Yaskawa INFORM job: apremTRJ2.JBI

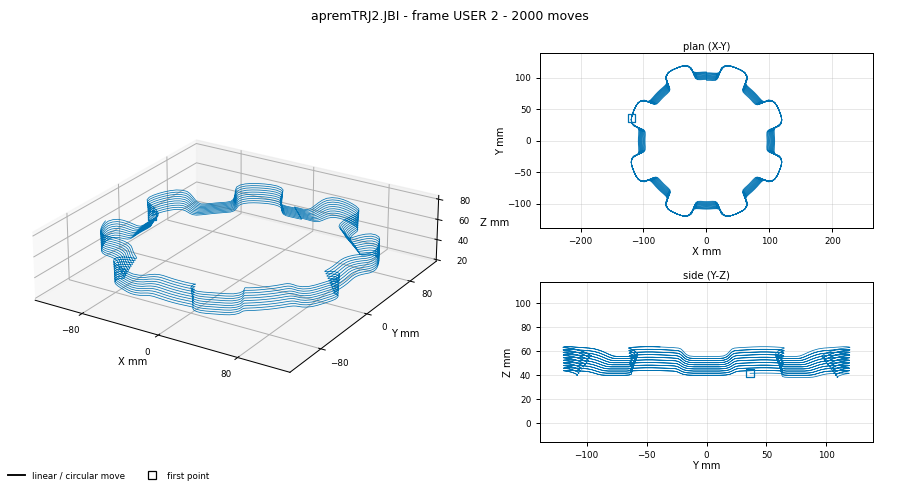
[picture p0: tool path of apremTRJ2.JBI in frame USER 2, 2000 of 2000 moves have a stored position in this frame; points joined in program order, loops and branches not executed]
/JOB
//NAME apremTRJ2
//POS
///NPOS 2000,0,0,0,0,0
///USER 2
///TOOL 1
///POSTYPE USER
///RECTAN
///RCONF 1,0,0,0,0,0,0,0,0,0,0,0,0,0,0,0,0,0,0,0,0,0,0,0
C00000=-119.072,36.353,41.582,179.9283,-0.7231,0.0000
C00001=-118.000,41.045,41.707,179.9989,-0.0034,0.0000
C00002=-116.380,45.594,41.789,179.9994,-0.0015,0.0000
C00003=-114.533,50.053,41.789,179.9993,-0.0015,0.0000
C00004=-112.462,54.416,41.707,179.9984,-0.0032,0.0000
C00005=-109.902,58.491,41.582,179.5393,-0.5620,0.0000
C00006=-106.611,61.626,41.458,179.6621,-0.2455,0.0000
C00007=-103.173,63.375,41.307,179.7307,-0.0735,0.0000
C00008=-100.060,63.578,41.020,-179.7213,-0.0197,0.0000
C00009=-97.017,63.208,40.437,-176.3792,-0.5593,0.0000
C00010=-94.156,62.962,39.673,-168.9691,-0.5777,0.0000
C00011=-91.471,63.401,38.921,-157.5827,5.7610,0.0000
C00012=-88.635,65.218,38.370,-153.3359,22.5360,0.0000
C00013=-85.107,69.037,38.148,-155.1849,27.9206,0.0000
C00014=-81.483,73.239,38.139,-154.7783,27.7766,0.0000
C00015=-77.473,77.473,38.145,-153.4608,26.5387,0.0000
C00016=-73.239,81.483,38.139,-152.2237,25.2220,0.0000
C00017=-69.037,85.107,38.148,-152.0801,24.8157,0.0000
C00018=-65.218,88.635,38.370,-157.4634,26.6637,0.0000
C00019=-63.401,91.471,38.921,-174.2390,22.4173,0.0000
C00020=-62.962,94.156,39.673,179.4223,11.0309,0.0000
C00021=-63.208,97.017,40.437,179.4407,3.6208,0.0000
C00022=-63.578,100.060,41.020,179.9803,0.2787,0.0000
C00023=-63.375,103.173,41.307,179.9265,-0.2693,0.0000
C00024=-61.626,106.611,41.458,179.7545,-0.3379,0.0000
C00025=-58.491,109.902,41.582,179.4380,-0.4607,0.0000
C00026=-54.416,112.462,41.707,179.9968,-0.0016,0.0000
C00027=-50.053,114.533,41.789,179.9985,-0.0007,0.0000
C00028=-45.594,116.380,41.789,179.9985,-0.0006,0.0000
C00029=-41.045,118.000,41.707,179.9966,-0.0011,0.0000
C00030=-36.353,119.072,41.582,179.2769,-0.0717,0.0000
C00031=-31.809,118.962,41.458,179.5875,0.0653,0.0000
C00032=-28.141,117.767,41.307,179.7576,0.1385,0.0000
C00033=-25.796,115.710,41.020,-179.8169,-0.2110,0.0000
C00034=-23.906,113.297,40.437,-177.8329,-2.9566,0.0000
C00035=-22.057,111.099,39.673,-172.5529,-8.2489,0.0000
C00036=-19.849,109.511,38.921,-160.0472,-12.4271,0.0000
C00037=-16.558,108.791,38.370,-147.0366,-3.5281,0.0000
C00038=-11.363,108.997,38.148,-144.9437,2.7334,0.0000
C00039=-5.830,109.405,38.139,-144.7966,2.2545,0.0000
C00040=0.000,109.564,38.145,-144.7664,0.0004,0.0000
C00041=0.000,108.284,39.935,-144.1032,0.0004,0.0000
C00042=5.713,108.130,39.927,-144.1335,-2.3009,0.0000
C00043=11.166,107.733,39.938,-144.2844,-2.6355,0.0000
C00044=16.317,107.567,40.182,-146.6500,4.4566,0.0000
C00045=19.551,108.390,40.791,-161.4224,13.0406,0.0000
C00046=21.713,110.141,41.623,-173.7880,7.6722,0.0000
C00047=23.528,112.556,42.474,-178.5737,2.1635,0.0000
C00048=25.385,115.220,43.124,179.5625,-0.5661,0.0000
C00049=27.691,117.522,43.446,179.0873,-0.5941,0.0000
C00050=31.383,118.911,43.616,179.2076,-0.1524,0.0000
C00051=36.015,119.134,43.755,179.1192,0.0737,0.0000
C00052=40.830,118.071,43.895,179.9841,0.0052,0.0000
C00053=45.521,116.408,43.987,179.9970,0.0012,0.0000
C00054=50.124,114.501,43.987,179.9971,0.0013,0.0000
C00055=54.618,112.360,43.895,179.9851,0.0076,0.0000
C00056=58.774,109.707,43.755,179.3251,0.5708,0.0000
C00057=61.891,106.274,43.616,179.5474,0.6680,0.0000
C00058=63.520,102.681,43.446,179.7747,1.0655,0.0000
C00059=63.523,99.422,43.124,-179.9091,0.7096,0.0000
C00060=62.953,96.226,42.474,179.4782,-2.5377,0.0000
C00061=62.528,93.235,41.623,178.9522,-9.7717,0.0000
C00062=62.818,90.468,40.791,-175.7744,-21.8723,0.0000
C00063=64.524,87.599,40.182,-157.6939,-27.4960,0.0000
C00064=68.283,84.074,39.938,-151.5889,-25.4475,0.0000
C00065=72.420,80.499,39.927,-151.6468,-25.7721,0.0000
C00066=76.568,76.568,39.935,-152.8969,-27.1036,0.0000
C00067=80.499,72.420,39.927,-154.2275,-28.3529,0.0000
C00068=84.074,68.282,39.938,-154.5518,-28.4103,0.0000
C00069=87.599,64.524,40.182,-152.5043,-22.3068,0.0000
C00070=90.468,62.818,40.791,-158.1277,-4.2256,0.0000
C00071=93.235,62.528,41.623,-170.2283,1.0478,0.0000
C00072=96.226,62.953,42.474,-177.4623,0.5218,0.0000
C00073=99.422,63.523,43.124,179.2904,-0.0909,0.0000
C00074=102.681,63.520,43.446,178.9345,0.2253,0.0000
C00075=106.274,61.891,43.616,179.3320,0.4526,0.0000
C00076=109.707,58.774,43.755,179.4292,0.6749,0.0000
C00077=112.360,54.618,43.895,179.9924,0.0149,0.0000
C00078=114.501,50.124,43.987,179.9987,0.0029,0.0000
C00079=116.408,45.521,43.987,179.9988,0.0030,0.0000
C00080=118.071,40.830,43.895,179.9948,0.0159,0.0000
C00081=119.134,36.015,43.755,179.9263,0.8808,0.0000
C00082=118.911,31.383,43.616,-179.8476,0.7924,0.0000
C00083=117.522,27.691,43.446,-179.4059,0.9127,0.0000
C00084=115.220,25.385,43.124,-179.4339,0.4375,0.0000
C00085=112.556,23.528,42.474,177.8365,-1.4263,0.0000
C00086=110.141,21.713,41.623,172.3278,-6.2120,0.0000
C00087=108.390,19.551,40.791,166.9594,-18.5776,0.0000
C00088=107.567,16.317,40.182,175.5434,-33.3500,0.0000
C00089=107.733,11.166,39.938,-177.3645,-35.7156,0.0000
C00090=108.130,5.713,39.927,-177.6991,-35.8665,0.0000
C00091=108.284,0.000,39.935,179.9996,-35.8968,0.0000
C00092=108.130,-5.713,39.927,177.6997,-35.8666,0.0000
C00093=107.733,-11.167,39.938,177.3658,-35.7155,0.0000
C00094=107.567,-16.317,40.182,-175.5442,-33.3502,0.0000
C00095=108.390,-19.551,40.791,-166.9594,-18.5776,0.0000
C00096=110.141,-21.713,41.623,-172.3278,-6.2120,0.0000
C00097=112.556,-23.528,42.474,-177.8365,-1.4263,0.0000
C00098=115.220,-25.385,43.124,179.4339,0.4375,0.0000
C00099=117.522,-27.691,43.446,179.4059,0.9127,0.0000
C00100=118.911,-31.383,43.616,179.8476,0.7924,0.0000
C00101=119.134,-36.015,43.755,-179.9263,0.8808,0.0000
C00102=118.071,-40.830,43.895,-179.9948,0.0159,0.0000
C00103=116.408,-45.521,43.987,-179.9988,0.0030,0.0000
C00104=114.501,-50.124,43.987,-179.9987,0.0029,0.0000
C00105=112.360,-54.618,43.895,-179.9924,0.0149,0.0000
C00106=109.707,-58.774,43.755,-179.4292,0.6749,0.0000
C00107=106.274,-61.891,43.616,-179.3320,0.4526,0.0000
C00108=102.681,-63.520,43.446,-178.9345,0.2253,0.0000
C00109=99.422,-63.523,43.124,-179.2904,-0.0909,0.0000
C00110=96.226,-62.953,42.474,177.4623,0.5218,0.0000
C00111=93.235,-62.528,41.623,170.2283,1.0478,0.0000
C00112=90.468,-62.818,40.791,158.1277,-4.2256,0.0000
C00113=87.599,-64.524,40.182,152.5040,-22.3061,0.0000
C00114=84.074,-68.283,39.938,154.5525,-28.4111,0.0000
C00115=80.499,-72.420,39.927,154.2279,-28.3532,0.0000
C00116=76.568,-76.568,39.935,152.8964,-27.1031,0.0000
C00117=72.420,-80.499,39.927,151.6471,-25.7725,0.0000
C00118=68.282,-84.074,39.938,151.5897,-25.4482,0.0000
C00119=64.524,-87.599,40.182,157.6932,-27.4957,0.0000
C00120=62.818,-90.468,40.791,175.7744,-21.8723,0.0000
C00121=62.528,-93.235,41.623,-178.9522,-9.7717,0.0000
C00122=62.953,-96.226,42.474,-179.4782,-2.5377,0.0000
C00123=63.523,-99.422,43.124,179.9091,0.7096,0.0000
C00124=63.520,-102.681,43.446,-179.7747,1.0655,0.0000
C00125=61.891,-106.274,43.616,-179.5474,0.6680,0.0000
C00126=58.774,-109.707,43.755,-179.3251,0.5708,0.0000
C00127=54.618,-112.360,43.895,-179.9851,0.0076,0.0000
C00128=50.124,-114.501,43.987,-179.9971,0.0013,0.0000
C00129=45.521,-116.408,43.987,-179.9970,0.0012,0.0000
C00130=40.830,-118.071,43.895,-179.9841,0.0052,0.0000
C00131=36.015,-119.134,43.755,-179.1192,0.0737,0.0000
C00132=31.383,-118.911,43.616,-179.2076,-0.1524,0.0000
C00133=27.691,-117.522,43.446,-179.0873,-0.5941,0.0000
C00134=25.385,-115.220,43.124,-179.5625,-0.5661,0.0000
C00135=23.528,-112.556,42.474,178.5737,2.1635,0.0000
C00136=21.713,-110.141,41.623,173.7880,7.6722,0.0000
C00137=19.551,-108.390,40.791,161.4224,13.0406,0.0000
C00138=16.317,-107.567,40.182,146.6500,4.4566,0.0000
C00139=11.166,-107.733,39.938,144.2844,-2.6355,0.0000
C00140=5.713,-108.130,39.927,144.1335,-2.3009,0.0000
C00141=0.000,-108.284,39.935,144.1032,0.0004,0.0000
C00142=0.000,-108.284,39.935,144.1032,0.0004,0.0000
C00143=-5.713,-108.130,39.927,144.1334,2.3003,0.0000
C00144=-11.167,-107.733,39.938,144.2845,2.6342,0.0000
C00145=-16.317,-107.567,40.182,146.6498,-4.4558,0.0000
C00146=-19.551,-108.390,40.791,161.4224,-13.0406,0.0000
C00147=-21.713,-110.141,41.623,173.7880,-7.6722,0.0000
C00148=-23.528,-112.556,42.474,178.5737,-2.1635,0.0000
C00149=-25.385,-115.220,43.124,-179.5625,0.5661,0.0000
C00150=-27.691,-117.522,43.446,-179.0873,0.5941,0.0000
C00151=-31.383,-118.911,43.616,-179.2076,0.1524,0.0000
C00152=-36.015,-119.134,43.755,-179.1192,-0.0737,0.0000
C00153=-40.830,-118.071,43.895,-179.9841,-0.0052,0.0000
C00154=-45.521,-116.408,43.987,-179.9970,-0.0012,0.0000
C00155=-50.124,-114.501,43.987,-179.9971,-0.0013,0.0000
C00156=-54.618,-112.360,43.895,-179.9851,-0.0076,0.0000
C00157=-58.774,-109.707,43.755,-179.3251,-0.5708,0.0000
C00158=-61.891,-106.274,43.616,-179.5474,-0.6680,0.0000
C00159=-63.520,-102.681,43.446,-179.7747,-1.0655,0.0000
C00160=-63.523,-99.422,43.124,179.9091,-0.7096,0.0000
C00161=-62.953,-96.226,42.474,-179.4782,2.5377,0.0000
C00162=-62.528,-93.235,41.623,-178.9522,9.7717,0.0000
C00163=-62.818,-90.468,40.791,175.7744,21.8723,0.0000
C00164=-64.524,-87.599,40.182,157.6939,27.4960,0.0000
C00165=-68.283,-84.074,39.938,151.5889,25.4475,0.0000
C00166=-72.420,-80.499,39.927,151.6468,25.7721,0.0000
C00167=-76.568,-76.568,39.935,152.8969,27.1036,0.0000
C00168=-80.499,-72.420,39.927,154.2275,28.3529,0.0000
C00169=-84.074,-68.282,39.938,154.5518,28.4103,0.0000
C00170=-87.599,-64.524,40.182,152.5043,22.3068,0.0000
C00171=-90.468,-62.818,40.791,158.1277,4.2256,0.0000
C00172=-93.235,-62.528,41.623,170.2283,-1.0478,0.0000
C00173=-96.226,-62.953,42.474,177.4623,-0.5218,0.0000
C00174=-99.422,-63.523,43.124,-179.2904,0.0909,0.0000
C00175=-102.681,-63.520,43.446,-178.9345,-0.2253,0.0000
C00176=-106.274,-61.891,43.616,-179.3320,-0.4526,0.0000
C00177=-109.707,-58.774,43.755,-179.4292,-0.6749,0.0000
C00178=-112.360,-54.618,43.895,-179.9924,-0.0149,0.0000
C00179=-114.501,-50.124,43.987,-179.9987,-0.0029,0.0000
C00180=-116.408,-45.521,43.987,-179.9988,-0.0030,0.0000
C00181=-118.071,-40.830,43.895,-179.9948,-0.0159,0.0000
C00182=-119.134,-36.015,43.755,-179.9263,-0.8808,0.0000
C00183=-118.911,-31.383,43.616,179.8476,-0.7924,0.0000
C00184=-117.522,-27.691,43.446,179.4059,-0.9127,0.0000
C00185=-115.220,-25.385,43.124,179.4339,-0.4375,0.0000
C00186=-112.556,-23.528,42.474,-177.8365,1.4263,0.0000
C00187=-110.141,-21.713,41.623,-172.3278,6.2120,0.0000
C00188=-108.390,-19.551,40.791,-166.9594,18.5776,0.0000
C00189=-107.567,-16.317,40.182,-175.5434,33.3500,0.0000
C00190=-107.733,-11.166,39.938,177.3645,35.7156,0.0000
C00191=-108.130,-5.713,39.927,177.6991,35.8665,0.0000
C00192=-108.284,0.000,39.935,-179.9996,35.8968,0.0000
C00193=-108.130,5.713,39.927,-177.6997,35.8666,0.0000
C00194=-107.733,11.167,39.938,-177.3658,35.7155,0.0000
C00195=-107.567,16.317,40.182,175.5442,33.3502,0.0000
C00196=-108.390,19.551,40.791,166.9594,18.5776,0.0000
C00197=-110.141,21.713,41.623,172.3278,6.2120,0.0000
C00198=-112.556,23.528,42.474,177.8365,1.4263,0.0000
C00199=-115.220,25.385,43.124,-179.4339,-0.4375,0.0000
C00200=-117.522,27.691,43.446,-179.4059,-0.9127,0.0000
C00201=-118.911,31.383,43.616,-179.8476,-0.7924,0.0000
C00202=-119.134,36.015,43.755,179.9263,-0.8808,0.0000
C00203=-118.071,40.830,43.895,179.9948,-0.0159,0.0000
C00204=-116.408,45.521,43.987,179.9988,-0.0030,0.0000
C00205=-114.501,50.124,43.987,179.9987,-0.0029,0.0000
C00206=-112.360,54.618,43.895,179.9924,-0.0149,0.0000
C00207=-109.707,58.774,43.755,179.4292,-0.6749,0.0000
C00208=-106.274,61.891,43.616,179.3320,-0.4526,0.0000
C00209=-102.681,63.520,43.446,178.9345,-0.2253,0.0000
C00210=-99.422,63.523,43.124,179.2904,0.0909,0.0000
C00211=-96.226,62.953,42.474,-177.4623,-0.5218,0.0000
C00212=-93.235,62.528,41.623,-170.2283,-1.0478,0.0000
C00213=-90.468,62.818,40.791,-158.1277,4.2256,0.0000
C00214=-87.599,64.524,40.182,-152.5040,22.3061,0.0000
C00215=-84.074,68.283,39.938,-154.5525,28.4111,0.0000
C00216=-80.499,72.420,39.927,-154.2279,28.3532,0.0000
C00217=-76.568,76.568,39.935,-152.8964,27.1031,0.0000
C00218=-72.420,80.499,39.927,-151.6471,25.7725,0.0000
C00219=-68.282,84.074,39.938,-151.5897,25.4482,0.0000
C00220=-64.524,87.599,40.182,-157.6932,27.4957,0.0000
C00221=-62.818,90.468,40.791,-175.7744,21.8723,0.0000
C00222=-62.528,93.235,41.623,178.9522,9.7717,0.0000
C00223=-62.953,96.226,42.474,179.4782,2.5377,0.0000
C00224=-63.523,99.422,43.124,-179.9091,-0.7096,0.0000
C00225=-63.520,102.681,43.446,179.7747,-1.0655,0.0000
C00226=-61.891,106.274,43.616,179.5474,-0.6680,0.0000
C00227=-58.774,109.707,43.755,179.3251,-0.5708,0.0000
C00228=-54.618,112.360,43.895,179.9851,-0.0076,0.0000
C00229=-50.124,114.501,43.987,179.9971,-0.0013,0.0000
C00230=-45.521,116.408,43.987,179.9970,-0.0012,0.0000
C00231=-40.830,118.071,43.895,179.9841,-0.0052,0.0000
C00232=-36.015,119.134,43.755,179.1192,-0.0737,0.0000
C00233=-31.383,118.911,43.616,179.2076,0.1524,0.0000
C00234=-27.691,117.522,43.446,179.0873,0.5941,0.0000
C00235=-25.385,115.220,43.124,179.5625,0.5661,0.0000
C00236=-23.528,112.556,42.474,-178.5737,-2.1635,0.0000
C00237=-21.713,110.141,41.623,-173.7880,-7.6722,0.0000
C00238=-19.551,108.390,40.791,-161.4224,-13.0406,0.0000
C00239=-16.317,107.567,40.182,-146.6498,-4.4558,0.0000
C00240=-11.167,107.733,39.938,-144.2845,2.6342,0.0000
C00241=-5.713,108.130,39.927,-144.1334,2.3003,0.0000
C00242=0.000,108.284,39.935,-144.1032,0.0004,0.0000
C00243=0.000,106.985,41.710,-143.5099,0.0004,0.0000
C00244=5.594,106.835,41.702,-143.5401,-2.3406,0.0000
C00245=10.967,106.449,41.714,-143.6958,-2.5164,0.0000
C00246=16.072,106.324,41.981,-146.3715,5.4141,0.0000
C00247=19.249,107.251,42.649,-162.9140,13.4061,0.0000
C00248=21.363,109.167,43.565,-174.8995,6.9770,0.0000
C00249=23.141,111.802,44.504,-179.1921,1.3529,0.0000
C00250=24.965,114.720,45.225,179.0571,-1.3592,0.0000
C00251=27.231,117.271,45.583,178.4751,-1.1175,0.0000
C00252=30.949,118.858,45.772,178.8291,-0.2647,0.0000
C00253=35.669,119.197,45.927,178.9615,0.0712,0.0000
C00254=40.611,118.143,46.083,179.9716,0.0092,0.0000
C00255=45.447,116.436,46.186,179.9955,0.0017,0.0000
C00256=50.197,114.469,46.186,179.9956,0.0019,0.0000
C00257=54.824,112.256,46.083,179.9734,0.0136,0.0000
C00258=59.063,109.507,45.927,179.2153,0.6841,0.0000
C00259=62.161,105.930,45.772,179.3591,1.0151,0.0000
C00260=63.668,102.179,45.583,179.7118,1.8682,0.0000
C00261=63.466,98.772,45.225,-179.7055,1.6276,0.0000
C00262=62.692,95.419,44.504,179.6145,-1.5278,0.0000
C00263=62.087,92.299,43.565,178.6584,-8.5110,0.0000
C00264=62.227,89.449,42.649,-177.2056,-21.1007,0.0000
C00265=63.818,86.547,41.981,-158.0362,-28.2502,0.0000
C00266=67.516,83.026,41.714,-151.1639,-26.0321,0.0000
C00267=71.588,79.499,41.702,-151.1291,-26.2693,0.0000
C00268=75.650,75.650,41.710,-152.3887,-27.6118,0.0000
C00269=79.499,71.588,41.702,-153.7304,-28.8707,0.0000
C00270=83.026,67.516,41.714,-153.9672,-28.8353,0.0000
C00271=86.547,63.818,41.981,-151.7501,-21.9645,0.0000
C00272=89.449,62.227,42.649,-158.8993,-2.7944,0.0000
C00273=92.299,62.087,43.565,-171.4890,1.3416,0.0000
C00274=95.419,62.692,44.504,-178.4722,0.3855,0.0000
C00275=98.772,63.466,45.225,178.3724,-0.2945,0.0000
C00276=102.179,63.668,45.583,178.1318,0.2882,0.0000
C00277=105.930,62.161,45.772,178.9849,0.6409,0.0000
C00278=109.507,59.063,45.927,179.3159,0.7847,0.0000
C00279=112.256,54.824,46.083,179.9864,0.0266,0.0000
C00280=114.469,50.197,46.186,179.9981,0.0044,0.0000
C00281=116.436,45.447,46.186,179.9983,0.0045,0.0000
C00282=118.143,40.611,46.083,179.9908,0.0284,0.0000
C00283=119.197,35.669,45.927,179.9288,1.0385,0.0000
C00284=118.858,30.949,45.772,-179.7353,1.1709,0.0000
C00285=117.271,27.231,45.583,-178.8825,1.5249,0.0000
C00286=114.720,24.965,45.225,-178.6408,0.9429,0.0000
C00287=111.802,23.141,44.504,178.6471,-0.8079,0.0000
C00288=109.167,21.363,43.565,173.0230,-5.1005,0.0000
C00289=107.251,19.249,42.649,166.5939,-17.0860,0.0000
C00290=106.324,16.072,41.981,174.5859,-33.6285,0.0000
C00291=106.449,10.967,41.714,-177.4836,-36.3042,0.0000
C00292=106.835,5.594,41.702,-177.6594,-36.4599,0.0000
C00293=106.985,0.000,41.710,179.9996,-36.4901,0.0000
C00294=106.835,-5.594,41.702,177.6600,-36.4599,0.0000
C00295=106.449,-10.967,41.714,177.4851,-36.3040,0.0000
C00296=106.324,-16.072,41.981,-174.5868,-33.6287,0.0000
C00297=107.251,-19.249,42.649,-166.5939,-17.0860,0.0000
C00298=109.167,-21.363,43.565,-173.0230,-5.1005,0.0000
C00299=111.802,-23.141,44.504,-178.6471,-0.8079,0.0000
C00300=114.720,-24.965,45.225,178.6408,0.9429,0.0000
C00301=117.271,-27.231,45.583,178.8825,1.5249,0.0000
C00302=118.858,-30.949,45.772,179.7353,1.1709,0.0000
C00303=119.197,-35.669,45.927,-179.9288,1.0385,0.0000
C00304=118.143,-40.611,46.083,-179.9908,0.0284,0.0000
C00305=116.436,-45.447,46.186,-179.9983,0.0045,0.0000
C00306=114.469,-50.197,46.186,-179.9981,0.0044,0.0000
C00307=112.256,-54.824,46.083,-179.9864,0.0266,0.0000
C00308=109.507,-59.063,45.927,-179.3159,0.7847,0.0000
C00309=105.930,-62.161,45.772,-178.9849,0.6409,0.0000
C00310=102.179,-63.668,45.583,-178.1318,0.2882,0.0000
C00311=98.772,-63.466,45.225,-178.3724,-0.2945,0.0000
C00312=95.419,-62.692,44.504,178.4722,0.3855,0.0000
C00313=92.299,-62.087,43.565,171.4890,1.3416,0.0000
C00314=89.449,-62.227,42.649,158.8993,-2.7944,0.0000
C00315=86.547,-63.818,41.981,151.7498,-21.9638,0.0000
C00316=83.026,-67.516,41.714,153.9679,-28.8361,0.0000
C00317=79.499,-71.588,41.702,153.7307,-28.8709,0.0000
C00318=75.650,-75.650,41.710,152.3882,-27.6113,0.0000
C00319=71.588,-79.499,41.702,151.1293,-26.2696,0.0000
C00320=67.516,-83.026,41.714,151.1647,-26.0328,0.0000
C00321=63.818,-86.547,41.981,158.0355,-28.2499,0.0000
C00322=62.227,-89.449,42.649,177.2056,-21.1007,0.0000
C00323=62.087,-92.299,43.565,-178.6584,-8.5110,0.0000
C00324=62.692,-95.419,44.504,-179.6145,-1.5278,0.0000
C00325=63.466,-98.772,45.225,179.7055,1.6276,0.0000
C00326=63.668,-102.179,45.583,-179.7118,1.8682,0.0000
C00327=62.161,-105.930,45.772,-179.3591,1.0151,0.0000
C00328=59.063,-109.507,45.927,-179.2153,0.6841,0.0000
C00329=54.824,-112.256,46.083,-179.9734,0.0136,0.0000
C00330=50.197,-114.469,46.186,-179.9956,0.0019,0.0000
C00331=45.447,-116.436,46.186,-179.9955,0.0017,0.0000
C00332=40.611,-118.143,46.083,-179.9716,0.0092,0.0000
C00333=35.669,-119.197,45.927,-178.9615,0.0712,0.0000
C00334=30.949,-118.858,45.772,-178.8291,-0.2647,0.0000
C00335=27.231,-117.271,45.583,-178.4751,-1.1175,0.0000
C00336=24.965,-114.720,45.225,-179.0571,-1.3592,0.0000
C00337=23.141,-111.802,44.504,179.1921,1.3529,0.0000
C00338=21.363,-109.167,43.565,174.8995,6.9770,0.0000
C00339=19.249,-107.251,42.649,162.9140,13.4061,0.0000
C00340=16.072,-106.324,41.981,146.3715,5.4141,0.0000
C00341=10.967,-106.449,41.714,143.6958,-2.5164,0.0000
C00342=5.594,-106.835,41.702,143.5401,-2.3406,0.0000
C00343=0.000,-106.985,41.710,143.5099,0.0004,0.0000
C00344=0.000,-106.985,41.710,143.5099,0.0004,0.0000
C00345=-5.594,-106.835,41.702,143.5401,2.3400,0.0000
C00346=-10.967,-106.449,41.714,143.6960,2.5149,0.0000
C00347=-16.072,-106.324,41.981,146.3713,-5.4132,0.0000
C00348=-19.249,-107.251,42.649,162.9140,-13.4061,0.0000
C00349=-21.363,-109.167,43.565,174.8995,-6.9770,0.0000
C00350=-23.141,-111.802,44.504,179.1921,-1.3529,0.0000
C00351=-24.965,-114.720,45.225,-179.0571,1.3592,0.0000
C00352=-27.231,-117.271,45.583,-178.4751,1.1175,0.0000
C00353=-30.949,-118.858,45.772,-178.8291,0.2647,0.0000
C00354=-35.669,-119.197,45.927,-178.9615,-0.0712,0.0000
C00355=-40.611,-118.143,46.083,-179.9716,-0.0092,0.0000
C00356=-45.447,-116.436,46.186,-179.9955,-0.0017,0.0000
C00357=-50.197,-114.469,46.186,-179.9956,-0.0019,0.0000
C00358=-54.824,-112.256,46.083,-179.9734,-0.0136,0.0000
C00359=-59.063,-109.507,45.927,-179.2153,-0.6841,0.0000
C00360=-62.161,-105.930,45.772,-179.3591,-1.0151,0.0000
C00361=-63.668,-102.179,45.583,-179.7118,-1.8682,0.0000
C00362=-63.466,-98.772,45.225,179.7055,-1.6276,0.0000
C00363=-62.692,-95.419,44.504,-179.6145,1.5278,0.0000
C00364=-62.087,-92.299,43.565,-178.6584,8.5110,0.0000
C00365=-62.227,-89.449,42.649,177.2056,21.1007,0.0000
C00366=-63.818,-86.547,41.981,158.0362,28.2502,0.0000
C00367=-67.516,-83.026,41.714,151.1639,26.0321,0.0000
C00368=-71.588,-79.499,41.702,151.1291,26.2693,0.0000
C00369=-75.650,-75.650,41.710,152.3887,27.6118,0.0000
C00370=-79.499,-71.588,41.702,153.7304,28.8707,0.0000
C00371=-83.026,-67.516,41.714,153.9672,28.8353,0.0000
C00372=-86.547,-63.818,41.981,151.7501,21.9645,0.0000
C00373=-89.449,-62.227,42.649,158.8993,2.7944,0.0000
C00374=-92.299,-62.087,43.565,171.4890,-1.3416,0.0000
C00375=-95.419,-62.692,44.504,178.4722,-0.3855,0.0000
C00376=-98.772,-63.466,45.225,-178.3724,0.2945,0.0000
C00377=-102.179,-63.668,45.583,-178.1318,-0.2882,0.0000
C00378=-105.930,-62.161,45.772,-178.9849,-0.6409,0.0000
C00379=-109.507,-59.063,45.927,-179.3159,-0.7847,0.0000
C00380=-112.256,-54.824,46.083,-179.9864,-0.0266,0.0000
C00381=-114.469,-50.197,46.186,-179.9981,-0.0044,0.0000
C00382=-116.436,-45.447,46.186,-179.9983,-0.0045,0.0000
C00383=-118.143,-40.611,46.083,-179.9908,-0.0284,0.0000
C00384=-119.197,-35.669,45.927,-179.9288,-1.0385,0.0000
C00385=-118.858,-30.949,45.772,179.7353,-1.1709,0.0000
C00386=-117.271,-27.231,45.583,178.8825,-1.5249,0.0000
C00387=-114.720,-24.965,45.225,178.6408,-0.9429,0.0000
C00388=-111.802,-23.141,44.504,-178.6471,0.8079,0.0000
C00389=-109.167,-21.363,43.565,-173.0230,5.1005,0.0000
C00390=-107.251,-19.249,42.649,-166.5939,17.0860,0.0000
C00391=-106.324,-16.072,41.981,-174.5859,33.6285,0.0000
C00392=-106.449,-10.967,41.714,177.4836,36.3042,0.0000
C00393=-106.835,-5.594,41.702,177.6594,36.4599,0.0000
C00394=-106.985,0.000,41.710,-179.9996,36.4901,0.0000
C00395=-106.835,5.594,41.702,-177.6600,36.4599,0.0000
C00396=-106.449,10.967,41.714,-177.4851,36.3040,0.0000
C00397=-106.324,16.072,41.981,174.5868,33.6287,0.0000
C00398=-107.251,19.249,42.649,166.5939,17.0860,0.0000
C00399=-109.167,21.363,43.565,173.0230,5.1005,0.0000
C00400=-111.802,23.141,44.504,178.6471,0.8079,0.0000
C00401=-114.720,24.965,45.225,-178.6408,-0.9429,0.0000
C00402=-117.271,27.231,45.583,-178.8825,-1.5249,0.0000
C00403=-118.858,30.949,45.772,-179.7353,-1.1709,0.0000
C00404=-119.197,35.669,45.927,179.9288,-1.0385,0.0000
C00405=-118.143,40.611,46.083,179.9908,-0.0284,0.0000
C00406=-116.436,45.447,46.186,179.9983,-0.0045,0.0000
C00407=-114.469,50.197,46.186,179.9981,-0.0044,0.0000
C00408=-112.256,54.824,46.083,179.9864,-0.0266,0.0000
C00409=-109.507,59.063,45.927,179.3159,-0.7847,0.0000
C00410=-105.930,62.161,45.772,178.9849,-0.6409,0.0000
C00411=-102.179,63.668,45.583,178.1318,-0.2882,0.0000
C00412=-98.772,63.466,45.225,178.3724,0.2945,0.0000
C00413=-95.419,62.692,44.504,-178.4722,-0.3855,0.0000
C00414=-92.299,62.087,43.565,-171.4890,-1.3416,0.0000
C00415=-89.449,62.227,42.649,-158.8993,2.7944,0.0000
C00416=-86.547,63.818,41.981,-151.7498,21.9638,0.0000
C00417=-83.026,67.516,41.714,-153.9679,28.8361,0.0000
C00418=-79.499,71.588,41.702,-153.7307,28.8709,0.0000
C00419=-75.650,75.650,41.710,-152.3882,27.6113,0.0000
C00420=-71.588,79.499,41.702,-151.1293,26.2696,0.0000
C00421=-67.516,83.026,41.714,-151.1647,26.0328,0.0000
C00422=-63.818,86.547,41.981,-158.0355,28.2499,0.0000
C00423=-62.227,89.449,42.649,-177.2056,21.1007,0.0000
C00424=-62.087,92.299,43.565,178.6584,8.5110,0.0000
C00425=-62.692,95.419,44.504,179.6145,1.5278,0.0000
C00426=-63.466,98.772,45.225,-179.7055,-1.6276,0.0000
C00427=-63.668,102.179,45.583,179.7118,-1.8682,0.0000
C00428=-62.161,105.930,45.772,179.3591,-1.0151,0.0000
C00429=-59.063,109.507,45.927,179.2153,-0.6841,0.0000
C00430=-54.824,112.256,46.083,179.9734,-0.0136,0.0000
C00431=-50.197,114.469,46.186,179.9956,-0.0019,0.0000
C00432=-45.447,116.436,46.186,179.9955,-0.0017,0.0000
C00433=-40.611,118.143,46.083,179.9716,-0.0092,0.0000
C00434=-35.669,119.197,45.927,178.9615,-0.0712,0.0000
C00435=-30.949,118.858,45.772,178.8291,0.2647,0.0000
C00436=-27.231,117.271,45.583,178.4751,1.1175,0.0000
C00437=-24.965,114.720,45.225,179.0571,1.3592,0.0000
C00438=-23.141,111.802,44.504,-179.1921,-1.3529,0.0000
C00439=-21.363,109.167,43.565,-174.8995,-6.9770,0.0000
C00440=-19.249,107.251,42.649,-162.9140,-13.4061,0.0000
C00441=-16.072,106.324,41.981,-146.3713,-5.4132,0.0000
C00442=-10.967,106.449,41.714,-143.6960,2.5149,0.0000
C00443=-5.594,106.835,41.702,-143.5401,2.3400,0.0000
C00444=0.000,106.985,41.710,-143.5099,0.0004,0.0000
C00445=0.000,105.668,43.472,-142.9821,0.0004,0.0000
C00446=5.474,105.523,43.464,-143.0123,-2.3744,0.0000
C00447=10.764,105.149,43.477,-143.1739,-2.3781,0.0000
C00448=15.823,105.065,43.767,-146.1991,6.3897,0.0000
C00449=18.943,106.095,44.495,-164.4703,13.5311,0.0000
C00450=21.007,108.178,45.497,-175.8811,6.2033,0.0000
C00451=22.749,111.035,46.529,-179.7006,0.5500,0.0000
C00452=24.538,114.212,47.323,178.6572,-2.1419,0.0000
C00453=26.763,117.017,47.718,177.9333,-1.6882,0.0000
C00454=30.507,118.805,47.927,178.4583,-0.3998,0.0000
C00455=35.318,119.261,48.097,178.8056,0.0643,0.0000
C00456=40.388,118.217,48.270,179.9591,0.0132,0.0000
C00457=45.371,116.466,48.385,179.9941,0.0023,0.0000
C00458=50.271,114.436,48.385,179.9942,0.0026,0.0000
C00459=55.033,112.151,48.270,179.9618,0.0196,0.0000
C00460=59.357,109.303,48.097,179.1099,0.7992,0.0000
C00461=62.436,105.579,47.927,179.1923,1.3729,0.0000
C00462=63.819,101.668,47.718,179.7321,2.6542,0.0000
C00463=63.409,98.111,47.323,-179.4345,2.4634,0.0000
C00464=62.427,94.599,46.529,179.8228,-0.6006,0.0000
C00465=61.639,91.348,45.497,178.5143,-7.2817,0.0000
C00466=61.626,88.415,44.495,-178.4920,-20.1360,0.0000
C00467=63.103,85.481,43.767,-158.4858,-28.9237,0.0000
C00468=66.740,81.963,43.477,-150.8013,-26.5705,0.0000
C00469=70.745,78.486,43.464,-150.6673,-26.7154,0.0000
C00470=74.719,74.719,43.472,-151.9342,-28.0663,0.0000
C00471=78.486,70.746,43.464,-153.2842,-29.3324,0.0000
C00472=81.963,66.740,43.477,-153.4287,-29.1978,0.0000
C00473=85.481,63.103,43.767,-151.0766,-21.5150,0.0000
C00474=88.415,61.626,44.495,-159.8640,-1.5080,0.0000
C00475=91.348,61.639,45.497,-172.7183,1.4857,0.0000
C00476=94.599,62.427,46.529,-179.3994,0.1772,0.0000
C00477=98.111,63.409,47.323,177.5366,-0.5655,0.0000
C00478=101.668,63.819,47.718,177.3458,0.2679,0.0000
C00479=105.579,62.436,47.927,178.6271,0.8077,0.0000
C00480=109.303,59.357,48.097,179.2008,0.8901,0.0000
C00481=112.151,55.033,48.270,179.9804,0.0382,0.0000
C00482=114.436,50.271,48.385,179.9974,0.0058,0.0000
C00483=116.466,45.371,48.385,179.9977,0.0059,0.0000
C00484=118.217,40.388,48.270,179.9868,0.0409,0.0000
C00485=119.261,35.318,48.097,179.9357,1.1944,0.0000
C00486=118.805,30.507,47.927,-179.6002,1.5417,0.0000
C00487=117.017,26.763,47.718,-178.3118,2.0667,0.0000
C00488=114.212,24.538,47.323,-177.8581,1.3428,0.0000
C00489=111.035,22.749,46.529,179.4500,-0.2994,0.0000
C00490=108.178,21.007,45.497,173.7967,-4.1189,0.0000
C00491=106.095,18.943,44.495,166.4689,-15.5297,0.0000
C00492=105.065,15.823,43.767,173.6103,-33.8009,0.0000
C00493=105.149,10.764,43.477,-177.6219,-36.8261,0.0000
C00494=105.523,5.474,43.464,-177.6256,-36.9877,0.0000
C00495=105.668,0.000,43.472,179.9996,-37.0179,0.0000
C00496=105.523,-5.474,43.464,177.6262,-36.9877,0.0000
C00497=105.149,-10.765,43.477,177.6234,-36.8259,0.0000
C00498=105.065,-15.823,43.767,-173.6112,-33.8012,0.0000
C00499=106.095,-18.943,44.495,-166.4689,-15.5297,0.0000
C00500=108.178,-21.007,45.497,-173.7967,-4.1189,0.0000
C00501=111.035,-22.749,46.529,-179.4500,-0.2994,0.0000
C00502=114.212,-24.538,47.323,177.8581,1.3428,0.0000
C00503=117.017,-26.763,47.718,178.3118,2.0667,0.0000
C00504=118.805,-30.507,47.927,179.6002,1.5417,0.0000
C00505=119.261,-35.318,48.097,-179.9357,1.1944,0.0000
C00506=118.217,-40.388,48.270,-179.9868,0.0409,0.0000
C00507=116.466,-45.371,48.385,-179.9977,0.0059,0.0000
C00508=114.436,-50.271,48.385,-179.9974,0.0058,0.0000
C00509=112.151,-55.033,48.270,-179.9804,0.0382,0.0000
C00510=109.303,-59.357,48.097,-179.2008,0.8901,0.0000
C00511=105.579,-62.436,47.927,-178.6271,0.8077,0.0000
C00512=101.668,-63.819,47.718,-177.3458,0.2679,0.0000
C00513=98.111,-63.409,47.323,-177.5366,-0.5655,0.0000
C00514=94.599,-62.427,46.529,179.3994,0.1772,0.0000
C00515=91.348,-61.639,45.497,172.7183,1.4857,0.0000
C00516=88.415,-61.626,44.495,159.8640,-1.5080,0.0000
C00517=85.481,-63.103,43.767,151.0763,-21.5142,0.0000
C00518=81.963,-66.740,43.477,153.4295,-29.1987,0.0000
C00519=78.486,-70.745,43.464,153.2846,-29.3327,0.0000
C00520=74.719,-74.719,43.472,151.9337,-28.0658,0.0000
C00521=70.746,-78.486,43.464,150.6676,-26.7158,0.0000
C00522=66.740,-81.963,43.477,150.8022,-26.5713,0.0000
C00523=63.103,-85.481,43.767,158.4850,-28.9234,0.0000
C00524=61.626,-88.415,44.495,178.4920,-20.1360,0.0000
C00525=61.639,-91.348,45.497,-178.5143,-7.2817,0.0000
C00526=62.427,-94.599,46.529,-179.8228,-0.6006,0.0000
C00527=63.409,-98.111,47.323,179.4345,2.4634,0.0000
C00528=63.819,-101.668,47.718,-179.7321,2.6542,0.0000
C00529=62.436,-105.579,47.927,-179.1923,1.3729,0.0000
C00530=59.357,-109.303,48.097,-179.1099,0.7992,0.0000
C00531=55.033,-112.151,48.270,-179.9618,0.0196,0.0000
C00532=50.271,-114.436,48.385,-179.9942,0.0026,0.0000
C00533=45.371,-116.466,48.385,-179.9941,0.0023,0.0000
C00534=40.388,-118.217,48.270,-179.9591,0.0132,0.0000
C00535=35.318,-119.261,48.097,-178.8056,0.0643,0.0000
C00536=30.507,-118.805,47.927,-178.4583,-0.3998,0.0000
C00537=26.763,-117.017,47.718,-177.9333,-1.6882,0.0000
C00538=24.538,-114.212,47.323,-178.6572,-2.1419,0.0000
C00539=22.749,-111.035,46.529,179.7006,0.5500,0.0000
C00540=21.007,-108.178,45.497,175.8811,6.2033,0.0000
C00541=18.943,-106.095,44.495,164.4703,13.5311,0.0000
C00542=15.823,-105.065,43.767,146.1991,6.3897,0.0000
C00543=10.764,-105.149,43.477,143.1739,-2.3781,0.0000
C00544=5.474,-105.523,43.464,143.0123,-2.3744,0.0000
C00545=0.000,-105.668,43.472,142.9821,0.0004,0.0000
C00546=0.000,-105.668,43.472,142.9821,0.0004,0.0000
C00547=-5.474,-105.523,43.464,143.0123,2.3738,0.0000
C00548=-10.765,-105.149,43.477,143.1741,2.3766,0.0000
C00549=-15.823,-105.065,43.767,146.1988,-6.3888,0.0000
C00550=-18.943,-106.095,44.495,164.4703,-13.5311,0.0000
C00551=-21.007,-108.178,45.497,175.8811,-6.2033,0.0000
C00552=-22.749,-111.035,46.529,179.7006,-0.5500,0.0000
C00553=-24.538,-114.212,47.323,-178.6572,2.1419,0.0000
C00554=-26.763,-117.017,47.718,-177.9333,1.6882,0.0000
C00555=-30.507,-118.805,47.927,-178.4583,0.3998,0.0000
C00556=-35.318,-119.261,48.097,-178.8056,-0.0643,0.0000
C00557=-40.388,-118.217,48.270,-179.9591,-0.0132,0.0000
C00558=-45.371,-116.466,48.385,-179.9941,-0.0023,0.0000
C00559=-50.271,-114.436,48.385,-179.9942,-0.0026,0.0000
C00560=-55.033,-112.151,48.270,-179.9618,-0.0196,0.0000
C00561=-59.357,-109.303,48.097,-179.1099,-0.7992,0.0000
C00562=-62.436,-105.579,47.927,-179.1923,-1.3729,0.0000
C00563=-63.819,-101.668,47.718,-179.7321,-2.6542,0.0000
C00564=-63.409,-98.111,47.323,179.4345,-2.4634,0.0000
C00565=-62.427,-94.599,46.529,-179.8228,0.6006,0.0000
C00566=-61.639,-91.348,45.497,-178.5143,7.2817,0.0000
C00567=-61.626,-88.415,44.495,178.4920,20.1360,0.0000
C00568=-63.103,-85.481,43.767,158.4858,28.9237,0.0000
C00569=-66.740,-81.963,43.477,150.8013,26.5705,0.0000
C00570=-70.745,-78.486,43.464,150.6673,26.7154,0.0000
C00571=-74.719,-74.719,43.472,151.9342,28.0663,0.0000
C00572=-78.486,-70.746,43.464,153.2842,29.3324,0.0000
C00573=-81.963,-66.740,43.477,153.4287,29.1978,0.0000
C00574=-85.481,-63.103,43.767,151.0766,21.5150,0.0000
C00575=-88.415,-61.626,44.495,159.8640,1.5080,0.0000
C00576=-91.348,-61.639,45.497,172.7183,-1.4857,0.0000
C00577=-94.599,-62.427,46.529,179.3994,-0.1772,0.0000
C00578=-98.111,-63.409,47.323,-177.5366,0.5655,0.0000
C00579=-101.668,-63.819,47.718,-177.3458,-0.2679,0.0000
C00580=-105.579,-62.436,47.927,-178.6271,-0.8077,0.0000
C00581=-109.303,-59.357,48.097,-179.2008,-0.8901,0.0000
C00582=-112.151,-55.033,48.270,-179.9804,-0.0382,0.0000
C00583=-114.436,-50.271,48.385,-179.9974,-0.0058,0.0000
C00584=-116.466,-45.371,48.385,-179.9977,-0.0059,0.0000
C00585=-118.217,-40.388,48.270,-179.9868,-0.0409,0.0000
C00586=-119.261,-35.318,48.097,-179.9357,-1.1944,0.0000
C00587=-118.805,-30.507,47.927,179.6002,-1.5417,0.0000
C00588=-117.017,-26.763,47.718,178.3118,-2.0667,0.0000
C00589=-114.212,-24.538,47.323,177.8581,-1.3428,0.0000
C00590=-111.035,-22.749,46.529,-179.4500,0.2994,0.0000
C00591=-108.178,-21.007,45.497,-173.7967,4.1189,0.0000
C00592=-106.095,-18.943,44.495,-166.4689,15.5297,0.0000
C00593=-105.065,-15.823,43.767,-173.6103,33.8009,0.0000
C00594=-105.149,-10.764,43.477,177.6219,36.8261,0.0000
C00595=-105.523,-5.474,43.464,177.6256,36.9877,0.0000
C00596=-105.668,0.000,43.472,-179.9996,37.0179,0.0000
C00597=-105.523,5.474,43.464,-177.6262,36.9877,0.0000
C00598=-105.149,10.765,43.477,-177.6234,36.8259,0.0000
C00599=-105.065,15.823,43.767,173.6112,33.8012,0.0000
C00600=-106.095,18.943,44.495,166.4689,15.5297,0.0000
C00601=-108.178,21.007,45.497,173.7967,4.1189,0.0000
C00602=-111.035,22.749,46.529,179.4500,0.2994,0.0000
C00603=-114.212,24.538,47.323,-177.8581,-1.3428,0.0000
C00604=-117.017,26.763,47.718,-178.3118,-2.0667,0.0000
C00605=-118.805,30.507,47.927,-179.6002,-1.5417,0.0000
C00606=-119.261,35.318,48.097,179.9357,-1.1944,0.0000
C00607=-118.217,40.388,48.270,179.9868,-0.0409,0.0000
C00608=-116.466,45.371,48.385,179.9977,-0.0059,0.0000
C00609=-114.436,50.271,48.385,179.9974,-0.0058,0.0000
C00610=-112.151,55.033,48.270,179.9804,-0.0382,0.0000
C00611=-109.303,59.357,48.097,179.2008,-0.8901,0.0000
C00612=-105.579,62.436,47.927,178.6271,-0.8077,0.0000
C00613=-101.668,63.819,47.718,177.3458,-0.2679,0.0000
C00614=-98.111,63.409,47.323,177.5366,0.5655,0.0000
C00615=-94.599,62.427,46.529,-179.3994,-0.1772,0.0000
C00616=-91.348,61.639,45.497,-172.7183,-1.4857,0.0000
C00617=-88.415,61.626,44.495,-159.8640,1.5080,0.0000
C00618=-85.481,63.103,43.767,-151.0763,21.5142,0.0000
C00619=-81.963,66.740,43.477,-153.4295,29.1987,0.0000
C00620=-78.486,70.745,43.464,-153.2846,29.3327,0.0000
C00621=-74.719,74.719,43.472,-151.9337,28.0658,0.0000
C00622=-70.746,78.486,43.464,-150.6676,26.7158,0.0000
C00623=-66.740,81.963,43.477,-150.8022,26.5713,0.0000
C00624=-63.103,85.481,43.767,-158.4850,28.9234,0.0000
C00625=-61.626,88.415,44.495,-178.4920,20.1360,0.0000
C00626=-61.639,91.348,45.497,178.5143,7.2817,0.0000
C00627=-62.427,94.599,46.529,179.8228,0.6006,0.0000
C00628=-63.409,98.111,47.323,-179.4345,-2.4634,0.0000
C00629=-63.819,101.668,47.718,179.7321,-2.6542,0.0000
C00630=-62.436,105.579,47.927,179.1923,-1.3729,0.0000
C00631=-59.357,109.303,48.097,179.1099,-0.7992,0.0000
C00632=-55.033,112.151,48.270,179.9618,-0.0196,0.0000
C00633=-50.271,114.436,48.385,179.9942,-0.0026,0.0000
C00634=-45.371,116.466,48.385,179.9941,-0.0023,0.0000
C00635=-40.388,118.217,48.270,179.9591,-0.0132,0.0000
C00636=-35.318,119.261,48.097,178.8056,-0.0643,0.0000
C00637=-30.507,118.805,47.927,178.4583,0.3998,0.0000
C00638=-26.763,117.017,47.718,177.9333,1.6882,0.0000
C00639=-24.538,114.212,47.323,178.6572,2.1419,0.0000
C00640=-22.749,111.035,46.529,-179.7006,-0.5500,0.0000
C00641=-21.007,108.178,45.497,-175.8811,-6.2033,0.0000
C00642=-18.943,106.095,44.495,-164.4703,-13.5311,0.0000
C00643=-15.823,105.065,43.767,-146.1988,-6.3888,0.0000
C00644=-10.765,105.149,43.477,-143.1741,2.3766,0.0000
C00645=-5.474,105.523,43.464,-143.0123,2.3738,0.0000
C00646=0.000,105.668,43.472,-142.9821,0.0004,0.0000
C00647=0.000,104.336,45.223,-142.5164,0.0004,0.0000
C00648=5.352,104.196,45.214,-142.5464,-2.4024,0.0000
C00649=10.560,103.833,45.228,-142.7151,-2.2217,0.0000
C00650=15.572,103.790,45.543,-146.1303,7.3717,0.0000
C00651=18.632,104.926,46.333,-166.0428,13.4333,0.0000
C00652=20.647,107.176,47.422,-176.7352,5.3847,0.0000
C00653=22.351,110.258,48.548,179.8865,-0.2274,0.0000
C00654=24.105,113.696,49.417,178.3499,-2.8948,0.0000
C00655=26.289,116.758,49.850,177.4682,-2.2858,0.0000
C00656=30.058,118.751,50.080,178.1009,-0.5547,0.0000
C00657=34.961,119.326,50.267,178.6533,0.0534,0.0000
C00658=40.162,118.292,50.457,179.9469,0.0170,0.0000
C00659=45.294,116.495,50.583,179.9927,0.0028,0.0000
C00660=50.347,114.402,50.583,179.9929,0.0032,0.0000
C00661=55.246,112.044,50.457,179.9504,0.0255,0.0000
C00662=59.655,109.097,50.267,179.0099,0.9146,0.0000
C00663=62.715,105.224,50.080,179.0490,1.7351,0.0000
C00664=63.972,101.150,49.850,179.8257,3.4046,0.0000
C00665=63.351,97.440,49.417,-179.1185,3.2124,0.0000
C00666=62.159,93.769,48.548,-179.9194,0.2411,0.0000
C00667=61.185,90.384,47.422,178.4926,-6.1066,0.0000
C00668=61.019,87.369,46.333,-179.6076,-19.0155,0.0000
C00669=62.380,84.402,45.543,-159.0366,-29.5140,0.0000
C00670=65.954,80.888,45.228,-150.4984,-27.0645,0.0000
C00671=69.893,77.462,45.214,-150.2590,-27.1128,0.0000
C00672=73.777,73.777,45.223,-151.5310,-28.4695,0.0000
C00673=77.462,69.893,45.214,-152.8869,-29.7407,0.0000
C00674=80.888,65.954,45.228,-152.9347,-29.5006,0.0000
C00675=84.402,62.380,45.543,-150.4862,-20.9643,0.0000
C00676=87.369,61.019,46.333,-160.9845,-0.3924,0.0000
C00677=90.384,61.185,47.422,-173.8934,1.5074,0.0000
C00678=93.769,62.159,48.548,179.7589,-0.0806,0.0000
C00679=97.440,63.351,49.417,176.7876,-0.8815,0.0000
C00680=101.150,63.972,49.850,176.5954,0.1743,0.0000
C00681=105.224,62.715,50.080,178.2649,0.9510,0.0000
C00682=109.097,59.655,50.267,179.0854,0.9901,0.0000
C00683=112.044,55.246,50.457,179.9745,0.0496,0.0000
C00684=114.402,50.347,50.583,179.9968,0.0071,0.0000
C00685=116.495,45.294,50.583,179.9972,0.0073,0.0000
C00686=118.292,40.162,50.457,179.9830,0.0531,0.0000
C00687=119.326,34.961,50.267,179.9466,1.3467,0.0000
C00688=118.751,30.058,50.080,-179.4453,1.8991,0.0000
C00689=116.758,26.289,49.850,-177.7142,2.5318,0.0000
C00690=113.696,24.105,49.417,-177.1052,1.6501,0.0000
C00691=110.258,22.351,48.548,-179.7726,0.1135,0.0000
C00692=107.176,20.647,47.422,174.6153,-3.2648,0.0000
C00693=104.926,18.632,46.333,166.5667,-13.9572,0.0000
C00694=103.790,15.572,45.543,172.6283,-33.8697,0.0000
C00695=103.833,10.560,45.228,-177.7783,-37.2849,0.0000
C00696=104.196,5.352,45.214,-177.5976,-37.4536,0.0000
C00697=104.336,0.000,45.223,179.9996,-37.4836,0.0000
C00698=104.196,-5.352,45.214,177.5982,-37.4537,0.0000
C00699=103.833,-10.560,45.228,177.7800,-37.2848,0.0000
C00700=103.790,-15.572,45.543,-172.6292,-33.8700,0.0000
C00701=104.926,-18.632,46.333,-166.5667,-13.9572,0.0000
C00702=107.176,-20.647,47.422,-174.6153,-3.2648,0.0000
C00703=110.258,-22.351,48.548,179.7726,0.1135,0.0000
C00704=113.696,-24.105,49.417,177.1052,1.6501,0.0000
C00705=116.758,-26.289,49.850,177.7142,2.5318,0.0000
C00706=118.751,-30.058,50.080,179.4453,1.8991,0.0000
C00707=119.326,-34.961,50.267,-179.9466,1.3467,0.0000
C00708=118.292,-40.162,50.457,-179.9830,0.0531,0.0000
C00709=116.495,-45.294,50.583,-179.9972,0.0073,0.0000
C00710=114.402,-50.347,50.583,-179.9968,0.0071,0.0000
C00711=112.044,-55.246,50.457,-179.9745,0.0496,0.0000
C00712=109.097,-59.655,50.267,-179.0854,0.9901,0.0000
C00713=105.224,-62.715,50.080,-178.2649,0.9510,0.0000
C00714=101.150,-63.972,49.850,-176.5954,0.1743,0.0000
C00715=97.440,-63.351,49.417,-176.7876,-0.8815,0.0000
C00716=93.769,-62.159,48.548,-179.7589,-0.0806,0.0000
C00717=90.384,-61.185,47.422,173.8934,1.5074,0.0000
C00718=87.369,-61.019,46.333,160.9845,-0.3924,0.0000
C00719=84.402,-62.380,45.543,150.4860,-20.9634,0.0000
C00720=80.888,-65.954,45.228,152.9355,-29.5016,0.0000
C00721=77.462,-69.893,45.214,152.8872,-29.7410,0.0000
C00722=73.777,-73.777,45.223,151.5305,-28.4690,0.0000
C00723=69.893,-77.462,45.214,150.2593,-27.1131,0.0000
C00724=65.954,-80.888,45.228,150.4994,-27.0653,0.0000
C00725=62.380,-84.402,45.543,159.0357,-29.5138,0.0000
C00726=61.019,-87.369,46.333,179.6076,-19.0155,0.0000
C00727=61.185,-90.384,47.422,-178.4926,-6.1066,0.0000
C00728=62.159,-93.769,48.548,179.9194,0.2411,0.0000
C00729=63.351,-97.440,49.417,179.1185,3.2124,0.0000
C00730=63.972,-101.150,49.850,-179.8257,3.4046,0.0000
C00731=62.715,-105.224,50.080,-179.0490,1.7351,0.0000
C00732=59.655,-109.097,50.267,-179.0099,0.9146,0.0000
C00733=55.246,-112.044,50.457,-179.9504,0.0255,0.0000
C00734=50.347,-114.402,50.583,-179.9929,0.0032,0.0000
C00735=45.294,-116.495,50.583,-179.9927,0.0028,0.0000
C00736=40.162,-118.292,50.457,-179.9469,0.0170,0.0000
C00737=34.961,-119.326,50.267,-178.6533,0.0534,0.0000
C00738=30.058,-118.751,50.080,-178.1009,-0.5547,0.0000
C00739=26.289,-116.758,49.850,-177.4682,-2.2858,0.0000
C00740=24.105,-113.696,49.417,-178.3499,-2.8948,0.0000
C00741=22.351,-110.258,48.548,-179.8865,-0.2274,0.0000
C00742=20.647,-107.176,47.422,176.7352,5.3847,0.0000
C00743=18.632,-104.926,46.333,166.0428,13.4333,0.0000
C00744=15.572,-103.790,45.543,146.1303,7.3717,0.0000
C00745=10.560,-103.833,45.228,142.7151,-2.2217,0.0000
C00746=5.352,-104.196,45.214,142.5464,-2.4024,0.0000
C00747=0.000,-104.336,45.223,142.5164,0.0004,0.0000
C00748=0.000,-104.336,45.223,142.5164,0.0004,0.0000
C00749=-5.352,-104.196,45.214,142.5463,2.4018,0.0000
C00750=-10.560,-103.833,45.228,142.7152,2.2200,0.0000
C00751=-15.572,-103.790,45.543,146.1300,-7.3708,0.0000
C00752=-18.632,-104.926,46.333,166.0428,-13.4333,0.0000
C00753=-20.647,-107.176,47.422,176.7352,-5.3847,0.0000
C00754=-22.351,-110.258,48.548,-179.8865,0.2274,0.0000
C00755=-24.105,-113.696,49.417,-178.3499,2.8948,0.0000
C00756=-26.289,-116.758,49.850,-177.4682,2.2858,0.0000
C00757=-30.058,-118.751,50.080,-178.1009,0.5547,0.0000
C00758=-34.961,-119.326,50.267,-178.6533,-0.0534,0.0000
C00759=-40.162,-118.292,50.457,-179.9469,-0.0170,0.0000
C00760=-45.294,-116.495,50.583,-179.9927,-0.0028,0.0000
C00761=-50.347,-114.402,50.583,-179.9929,-0.0032,0.0000
C00762=-55.246,-112.044,50.457,-179.9504,-0.0255,0.0000
C00763=-59.655,-109.097,50.267,-179.0099,-0.9146,0.0000
C00764=-62.715,-105.224,50.080,-179.0490,-1.7351,0.0000
C00765=-63.972,-101.150,49.850,-179.8257,-3.4046,0.0000
C00766=-63.351,-97.440,49.417,179.1185,-3.2124,0.0000
C00767=-62.159,-93.769,48.548,179.9194,-0.2411,0.0000
C00768=-61.185,-90.384,47.422,-178.4926,6.1066,0.0000
C00769=-61.019,-87.369,46.333,179.6076,19.0155,0.0000
C00770=-62.380,-84.402,45.543,159.0366,29.5140,0.0000
C00771=-65.954,-80.888,45.228,150.4984,27.0645,0.0000
C00772=-69.893,-77.462,45.214,150.2590,27.1128,0.0000
C00773=-73.777,-73.777,45.223,151.5310,28.4695,0.0000
C00774=-77.462,-69.893,45.214,152.8869,29.7407,0.0000
C00775=-80.888,-65.954,45.228,152.9347,29.5006,0.0000
C00776=-84.402,-62.380,45.543,150.4862,20.9643,0.0000
C00777=-87.369,-61.019,46.333,160.9845,0.3924,0.0000
C00778=-90.384,-61.185,47.422,173.8934,-1.5074,0.0000
C00779=-93.769,-62.159,48.548,-179.7589,0.0806,0.0000
C00780=-97.440,-63.351,49.417,-176.7876,0.8815,0.0000
C00781=-101.150,-63.972,49.850,-176.5954,-0.1743,0.0000
C00782=-105.224,-62.715,50.080,-178.2649,-0.9510,0.0000
C00783=-109.097,-59.655,50.267,-179.0854,-0.9901,0.0000
C00784=-112.044,-55.246,50.457,-179.9745,-0.0496,0.0000
C00785=-114.402,-50.347,50.583,-179.9968,-0.0071,0.0000
C00786=-116.495,-45.294,50.583,-179.9972,-0.0073,0.0000
C00787=-118.292,-40.162,50.457,-179.9830,-0.0531,0.0000
C00788=-119.326,-34.961,50.267,-179.9466,-1.3467,0.0000
C00789=-118.751,-30.058,50.080,179.4453,-1.8991,0.0000
C00790=-116.758,-26.289,49.850,177.7142,-2.5318,0.0000
C00791=-113.696,-24.105,49.417,177.1052,-1.6501,0.0000
C00792=-110.258,-22.351,48.548,179.7726,-0.1135,0.0000
C00793=-107.176,-20.647,47.422,-174.6153,3.2648,0.0000
C00794=-104.926,-18.632,46.333,-166.5667,13.9572,0.0000
C00795=-103.790,-15.572,45.543,-172.6283,33.8697,0.0000
C00796=-103.833,-10.560,45.228,177.7783,37.2849,0.0000
C00797=-104.196,-5.352,45.214,177.5976,37.4536,0.0000
C00798=-104.336,0.000,45.223,-179.9996,37.4836,0.0000
C00799=-104.196,5.352,45.214,-177.5982,37.4537,0.0000
C00800=-103.833,10.560,45.228,-177.7800,37.2848,0.0000
C00801=-103.790,15.572,45.543,172.6292,33.8700,0.0000
C00802=-104.926,18.632,46.333,166.5667,13.9572,0.0000
C00803=-107.176,20.647,47.422,174.6153,3.2648,0.0000
C00804=-110.258,22.351,48.548,-179.7726,-0.1135,0.0000
C00805=-113.696,24.105,49.417,-177.1052,-1.6501,0.0000
C00806=-116.758,26.289,49.850,-177.7142,-2.5318,0.0000
C00807=-118.751,30.058,50.080,-179.4453,-1.8991,0.0000
C00808=-119.326,34.961,50.267,179.9466,-1.3467,0.0000
C00809=-118.292,40.162,50.457,179.9830,-0.0531,0.0000
C00810=-116.495,45.294,50.583,179.9972,-0.0073,0.0000
C00811=-114.402,50.347,50.583,179.9968,-0.0071,0.0000
C00812=-112.044,55.246,50.457,179.9745,-0.0496,0.0000
C00813=-109.097,59.655,50.267,179.0854,-0.9901,0.0000
C00814=-105.224,62.715,50.080,178.2649,-0.9510,0.0000
C00815=-101.150,63.972,49.850,176.5954,-0.1743,0.0000
C00816=-97.440,63.351,49.417,176.7876,0.8815,0.0000
C00817=-93.769,62.159,48.548,179.7589,0.0806,0.0000
C00818=-90.384,61.185,47.422,-173.8934,-1.5074,0.0000
C00819=-87.369,61.019,46.333,-160.9845,0.3924,0.0000
C00820=-84.402,62.380,45.543,-150.4860,20.9634,0.0000
C00821=-80.888,65.954,45.228,-152.9355,29.5016,0.0000
C00822=-77.462,69.893,45.214,-152.8872,29.7410,0.0000
C00823=-73.777,73.777,45.223,-151.5305,28.4690,0.0000
C00824=-69.893,77.462,45.214,-150.2593,27.1131,0.0000
C00825=-65.954,80.888,45.228,-150.4994,27.0653,0.0000
C00826=-62.380,84.402,45.543,-159.0357,29.5138,0.0000
C00827=-61.019,87.369,46.333,-179.6076,19.0155,0.0000
C00828=-61.185,90.384,47.422,178.4926,6.1066,0.0000
C00829=-62.159,93.769,48.548,-179.9194,-0.2411,0.0000
C00830=-63.351,97.440,49.417,-179.1185,-3.2124,0.0000
C00831=-63.972,101.150,49.850,179.8257,-3.4046,0.0000
C00832=-62.715,105.224,50.080,179.0490,-1.7351,0.0000
C00833=-59.655,109.097,50.267,179.0099,-0.9146,0.0000
C00834=-55.246,112.044,50.457,179.9504,-0.0255,0.0000
C00835=-50.347,114.402,50.583,179.9929,-0.0032,0.0000
C00836=-45.294,116.495,50.583,179.9927,-0.0028,0.0000
C00837=-40.162,118.292,50.457,179.9469,-0.0170,0.0000
C00838=-34.961,119.326,50.267,178.6533,-0.0534,0.0000
C00839=-30.058,118.751,50.080,178.1009,0.5547,0.0000
C00840=-26.289,116.758,49.850,177.4682,2.2858,0.0000
C00841=-24.105,113.696,49.417,178.3499,2.8948,0.0000
C00842=-22.351,110.258,48.548,179.8865,0.2274,0.0000
C00843=-20.647,107.176,47.422,-176.7352,-5.3847,0.0000
C00844=-18.632,104.926,46.333,-166.0428,-13.4333,0.0000
C00845=-15.572,103.790,45.543,-146.1300,-7.3708,0.0000
C00846=-10.560,103.833,45.228,-142.7152,2.2200,0.0000
C00847=-5.352,104.196,45.214,-142.5463,2.4018,0.0000
C00848=0.000,104.336,45.223,-142.5164,0.0004,0.0000
C00849=0.000,102.991,46.964,-142.1093,0.0004,0.0000
C00850=5.229,102.855,46.955,-142.1391,-2.4246,0.0000
C00851=10.353,102.505,46.969,-142.3163,-2.0479,0.0000
C00852=15.318,102.503,47.308,-146.1630,8.3483,0.0000
C00853=18.319,103.744,48.162,-167.5891,13.1372,0.0000
C00854=20.283,106.163,49.341,-177.4697,4.5481,0.0000
C00855=21.949,109.472,50.563,179.5554,-0.9673,0.0000
C00856=23.667,113.175,51.509,178.1218,-3.6046,0.0000
C00857=25.809,116.497,51.981,177.0809,-2.8914,0.0000
C00858=29.604,118.696,52.232,177.7619,-0.7258,0.0000
C00859=34.600,119.391,52.436,178.5062,0.0387,0.0000
C00860=39.933,118.367,52.644,179.9350,0.0207,0.0000
C00861=45.216,116.525,52.781,179.9913,0.0033,0.0000
C00862=50.423,114.369,52.781,179.9915,0.0038,0.0000
C00863=55.461,111.935,52.644,179.9394,0.0313,0.0000
C00864=59.957,108.888,52.436,178.9162,1.0290,0.0000
C00865=62.998,104.864,52.232,178.9299,2.0957,0.0000
C00866=64.126,100.625,51.981,179.9804,4.1051,0.0000
C00867=63.292,96.762,51.509,-178.7765,3.8749,0.0000
C00868=61.888,92.928,50.563,-179.6303,0.9984,0.0000
C00869=60.727,89.411,49.341,178.5679,-5.0004,0.0000
C00870=60.405,86.311,48.162,179.4600,-17.7781,0.0000
C00871=61.649,83.312,47.308,-159.6822,-30.0191,0.0000
C00872=65.161,79.802,46.969,-150.2530,-27.5154,0.0000
C00873=69.032,76.427,46.955,-149.9020,-27.4632,0.0000
C00874=72.826,72.826,46.964,-151.1770,-28.8234,0.0000
C00875=76.427,69.032,46.955,-152.5364,-30.0977,0.0000
C00876=79.802,65.161,46.969,-152.4838,-29.7459,0.0000
C00877=83.312,61.649,47.309,-149.9811,-20.3186,0.0000
C00878=86.311,60.405,48.162,-162.2219,0.5400,0.0000
C00879=89.411,60.727,49.341,-174.9996,1.4321,0.0000
C00880=92.928,61.888,50.563,179.0016,-0.3697,0.0000
C00881=96.762,63.292,51.509,176.1251,-1.2235,0.0000
C00882=100.625,64.126,51.981,175.8949,0.0196,0.0000
C00883=104.864,62.998,52.232,177.9043,1.0701,0.0000
C00884=108.888,59.957,52.436,178.9710,1.0838,0.0000
C00885=111.935,55.461,52.644,179.9687,0.0606,0.0000
C00886=114.369,50.423,52.781,179.9962,0.0085,0.0000
C00887=116.525,45.216,52.781,179.9967,0.0087,0.0000
C00888=118.367,39.933,52.644,179.9793,0.0650,0.0000
C00889=119.391,34.600,52.436,179.9613,1.4938,0.0000
C00890=118.696,29.604,52.232,-179.2742,2.2381,0.0000
C00891=116.497,25.809,51.981,-177.1086,2.9191,0.0000
C00892=113.175,23.667,51.509,-176.3954,1.8782,0.0000
C00893=109.472,21.949,50.563,-179.0327,0.4446,0.0000
C00894=106.163,20.283,49.341,175.4519,-2.5303,0.0000
C00895=103.744,18.319,48.162,166.8628,-12.4109,0.0000
C00896=102.503,15.318,47.308,171.6517,-33.8370,0.0000
C00897=102.505,10.353,46.969,-177.9521,-37.6837,0.0000
C00898=102.855,5.229,46.955,-177.5754,-37.8609,0.0000
C00899=102.991,0.000,46.964,179.9996,-37.8907,0.0000
C00900=102.855,-5.229,46.955,177.5759,-37.8609,0.0000
C00901=102.505,-10.353,46.969,177.9538,-37.6835,0.0000
C00902=102.503,-15.318,47.309,-171.6525,-33.8374,0.0000
C00903=103.744,-18.319,48.162,-166.8628,-12.4109,0.0000
C00904=106.163,-20.283,49.341,-175.4519,-2.5303,0.0000
C00905=109.472,-21.949,50.563,179.0327,0.4446,0.0000
C00906=113.175,-23.667,51.509,176.3954,1.8782,0.0000
C00907=116.497,-25.809,51.981,177.1086,2.9191,0.0000
C00908=118.696,-29.604,52.232,179.2742,2.2381,0.0000
C00909=119.391,-34.600,52.436,-179.9613,1.4938,0.0000
C00910=118.367,-39.933,52.644,-179.9793,0.0650,0.0000
C00911=116.525,-45.216,52.781,-179.9967,0.0087,0.0000
C00912=114.369,-50.423,52.781,-179.9962,0.0085,0.0000
C00913=111.935,-55.461,52.644,-179.9687,0.0606,0.0000
C00914=108.888,-59.957,52.436,-178.9710,1.0838,0.0000
C00915=104.864,-62.998,52.232,-177.9043,1.0701,0.0000
C00916=100.625,-64.126,51.981,-175.8949,0.0196,0.0000
C00917=96.762,-63.292,51.509,-176.1251,-1.2235,0.0000
C00918=92.928,-61.888,50.563,-179.0016,-0.3697,0.0000
C00919=89.411,-60.727,49.341,174.9996,1.4321,0.0000
C00920=86.311,-60.405,48.162,162.2219,0.5400,0.0000
C00921=83.312,-61.649,47.308,149.9809,-20.3178,0.0000
C00922=79.802,-65.161,46.969,152.4846,-29.7470,0.0000
C00923=76.427,-69.032,46.955,152.5368,-30.0980,0.0000
C00924=72.826,-72.826,46.964,151.1766,-28.8230,0.0000
C00925=69.032,-76.427,46.955,149.9023,-27.4636,0.0000
C00926=65.161,-79.802,46.969,150.2541,-27.5162,0.0000
C00927=61.649,-83.312,47.309,159.6814,-30.0189,0.0000
C00928=60.405,-86.311,48.162,-179.4600,-17.7781,0.0000
C00929=60.727,-89.411,49.341,-178.5679,-5.0004,0.0000
C00930=61.888,-92.928,50.563,179.6303,0.9984,0.0000
C00931=63.292,-96.762,51.509,178.7765,3.8749,0.0000
C00932=64.126,-100.625,51.981,-179.9804,4.1051,0.0000
C00933=62.998,-104.864,52.232,-178.9299,2.0957,0.0000
C00934=59.957,-108.888,52.436,-178.9162,1.0290,0.0000
C00935=55.461,-111.935,52.644,-179.9394,0.0313,0.0000
C00936=50.423,-114.369,52.781,-179.9915,0.0038,0.0000
C00937=45.216,-116.525,52.781,-179.9913,0.0033,0.0000
C00938=39.933,-118.367,52.644,-179.9350,0.0207,0.0000
C00939=34.600,-119.391,52.436,-178.5062,0.0387,0.0000
C00940=29.604,-118.696,52.232,-177.7619,-0.7258,0.0000
C00941=25.809,-116.497,51.981,-177.0809,-2.8914,0.0000
C00942=23.667,-113.175,51.509,-178.1218,-3.6046,0.0000
C00943=21.949,-109.472,50.563,-179.5554,-0.9673,0.0000
C00944=20.283,-106.163,49.341,177.4697,4.5481,0.0000
C00945=18.319,-103.744,48.162,167.5891,13.1372,0.0000
C00946=15.318,-102.503,47.308,146.1630,8.3483,0.0000
C00947=10.353,-102.505,46.969,142.3163,-2.0479,0.0000
C00948=5.229,-102.855,46.955,142.1391,-2.4246,0.0000
C00949=0.000,-102.991,46.964,142.1093,0.0004,0.0000
C00950=0.000,-102.991,46.964,142.1093,0.0004,0.0000
C00951=-5.229,-102.855,46.955,142.1391,2.4241,0.0000
C00952=-10.353,-102.505,46.969,142.3165,2.0462,0.0000
C00953=-15.318,-102.503,47.309,146.1626,-8.3475,0.0000
C00954=-18.319,-103.744,48.162,167.5891,-13.1372,0.0000
C00955=-20.283,-106.163,49.341,177.4697,-4.5481,0.0000
C00956=-21.949,-109.472,50.563,-179.5554,0.9673,0.0000
C00957=-23.667,-113.175,51.509,-178.1218,3.6046,0.0000
C00958=-25.809,-116.497,51.981,-177.0809,2.8914,0.0000
C00959=-29.604,-118.696,52.232,-177.7619,0.7258,0.0000
C00960=-34.600,-119.391,52.436,-178.5062,-0.0387,0.0000
C00961=-39.933,-118.367,52.644,-179.9350,-0.0207,0.0000
C00962=-45.216,-116.525,52.781,-179.9913,-0.0033,0.0000
C00963=-50.423,-114.369,52.781,-179.9915,-0.0038,0.0000
C00964=-55.461,-111.935,52.644,-179.9394,-0.0313,0.0000
C00965=-59.957,-108.888,52.436,-178.9162,-1.0290,0.0000
C00966=-62.998,-104.864,52.232,-178.9299,-2.0957,0.0000
C00967=-64.126,-100.625,51.981,-179.9804,-4.1051,0.0000
C00968=-63.292,-96.762,51.509,178.7765,-3.8749,0.0000
C00969=-61.888,-92.928,50.563,179.6303,-0.9984,0.0000
C00970=-60.727,-89.411,49.341,-178.5679,5.0004,0.0000
C00971=-60.405,-86.311,48.162,-179.4600,17.7781,0.0000
C00972=-61.649,-83.312,47.308,159.6822,30.0191,0.0000
C00973=-65.161,-79.802,46.969,150.2530,27.5154,0.0000
C00974=-69.032,-76.427,46.955,149.9020,27.4632,0.0000
C00975=-72.826,-72.826,46.964,151.1770,28.8234,0.0000
C00976=-76.427,-69.032,46.955,152.5364,30.0977,0.0000
C00977=-79.802,-65.161,46.969,152.4838,29.7459,0.0000
C00978=-83.312,-61.649,47.309,149.9811,20.3186,0.0000
C00979=-86.311,-60.405,48.162,162.2219,-0.5400,0.0000
C00980=-89.411,-60.727,49.341,174.9996,-1.4321,0.0000
C00981=-92.928,-61.888,50.563,-179.0016,0.3697,0.0000
C00982=-96.762,-63.292,51.509,-176.1251,1.2235,0.0000
C00983=-100.625,-64.126,51.981,-175.8949,-0.0196,0.0000
C00984=-104.864,-62.998,52.232,-177.9043,-1.0701,0.0000
C00985=-108.888,-59.957,52.436,-178.9710,-1.0838,0.0000
C00986=-111.935,-55.461,52.644,-179.9687,-0.0606,0.0000
C00987=-114.369,-50.423,52.781,-179.9962,-0.0085,0.0000
C00988=-116.525,-45.216,52.781,-179.9967,-0.0087,0.0000
C00989=-118.367,-39.933,52.644,-179.9793,-0.0650,0.0000
C00990=-119.391,-34.600,52.436,-179.9613,-1.4938,0.0000
C00991=-118.696,-29.604,52.232,179.2742,-2.2381,0.0000
C00992=-116.497,-25.809,51.981,177.1086,-2.9191,0.0000
C00993=-113.175,-23.667,51.509,176.3954,-1.8782,0.0000
C00994=-109.472,-21.949,50.563,179.0327,-0.4446,0.0000
C00995=-106.163,-20.283,49.341,-175.4519,2.5303,0.0000
C00996=-103.744,-18.319,48.162,-166.8628,12.4109,0.0000
C00997=-102.503,-15.318,47.308,-171.6517,33.8370,0.0000
C00998=-102.505,-10.353,46.969,177.9521,37.6837,0.0000
C00999=-102.855,-5.229,46.955,177.5754,37.8609,0.0000
C01000=-102.991,0.000,46.964,-179.9996,37.8907,0.0000
C01001=-102.855,5.229,46.955,-177.5759,37.8609,0.0000
C01002=-102.505,10.353,46.969,-177.9538,37.6835,0.0000
C01003=-102.503,15.318,47.309,171.6525,33.8374,0.0000
C01004=-103.744,18.319,48.162,166.8628,12.4109,0.0000
C01005=-106.163,20.283,49.341,175.4519,2.5303,0.0000
C01006=-109.472,21.949,50.563,-179.0327,-0.4446,0.0000
C01007=-113.175,23.667,51.509,-176.3954,-1.8782,0.0000
C01008=-116.497,25.809,51.981,-177.1086,-2.9191,0.0000
C01009=-118.696,29.604,52.232,-179.2742,-2.2381,0.0000
C01010=-119.391,34.600,52.436,179.9613,-1.4938,0.0000
C01011=-118.367,39.933,52.644,179.9793,-0.0650,0.0000
C01012=-116.525,45.216,52.781,179.9967,-0.0087,0.0000
C01013=-114.369,50.423,52.781,179.9962,-0.0085,0.0000
C01014=-111.935,55.461,52.644,179.9687,-0.0606,0.0000
C01015=-108.888,59.957,52.436,178.9710,-1.0838,0.0000
C01016=-104.864,62.998,52.232,177.9043,-1.0701,0.0000
C01017=-100.625,64.126,51.981,175.8949,-0.0196,0.0000
C01018=-96.762,63.292,51.509,176.1251,1.2235,0.0000
C01019=-92.928,61.888,50.563,179.0016,0.3697,0.0000
C01020=-89.411,60.727,49.341,-174.9996,-1.4321,0.0000
C01021=-86.311,60.405,48.162,-162.2219,-0.5400,0.0000
C01022=-83.312,61.649,47.308,-149.9809,20.3178,0.0000
C01023=-79.802,65.161,46.969,-152.4846,29.7470,0.0000
C01024=-76.427,69.032,46.955,-152.5368,30.0980,0.0000
C01025=-72.826,72.826,46.964,-151.1766,28.8230,0.0000
C01026=-69.032,76.427,46.955,-149.9023,27.4636,0.0000
C01027=-65.161,79.802,46.969,-150.2541,27.5162,0.0000
C01028=-61.649,83.312,47.309,-159.6814,30.0189,0.0000
C01029=-60.405,86.311,48.162,179.4600,17.7781,0.0000
C01030=-60.727,89.411,49.341,178.5679,5.0004,0.0000
C01031=-61.888,92.928,50.563,-179.6303,-0.9984,0.0000
C01032=-63.292,96.762,51.509,-178.7765,-3.8749,0.0000
C01033=-64.126,100.625,51.981,179.9804,-4.1051,0.0000
C01034=-62.998,104.864,52.232,178.9299,-2.0957,0.0000
C01035=-59.957,108.888,52.436,178.9162,-1.0290,0.0000
C01036=-55.461,111.935,52.644,179.9394,-0.0313,0.0000
C01037=-50.423,114.369,52.781,179.9915,-0.0038,0.0000
C01038=-45.216,116.525,52.781,179.9913,-0.0033,0.0000
C01039=-39.933,118.367,52.644,179.9350,-0.0207,0.0000
C01040=-34.600,119.391,52.436,178.5062,-0.0387,0.0000
C01041=-29.604,118.696,52.232,177.7619,0.7258,0.0000
C01042=-25.809,116.497,51.981,177.0809,2.8914,0.0000
C01043=-23.667,113.175,51.509,178.1218,3.6046,0.0000
C01044=-21.949,109.472,50.563,179.5554,0.9673,0.0000
C01045=-20.283,106.163,49.341,-177.4697,-4.5481,0.0000
C01046=-18.319,103.744,48.162,-167.5891,-13.1372,0.0000
C01047=-15.318,102.503,47.309,-146.1626,-8.3475,0.0000
C01048=-10.353,102.505,46.969,-142.3165,2.0462,0.0000
C01049=-5.229,102.855,46.955,-142.1391,2.4241,0.0000
C01050=0.000,102.991,46.964,-142.1093,0.0004,0.0000
C01051=0.000,101.635,48.696,-141.7583,0.0003,0.0000
C01052=5.105,101.503,48.686,-141.7878,-2.4412,0.0000
C01053=10.144,101.164,48.701,-141.9749,-1.8579,0.0000
C01054=15.062,101.204,49.066,-146.2949,9.3079,0.0000
C01055=18.003,102.552,49.983,-169.0746,12.6714,0.0000
C01056=19.915,105.141,51.254,-178.0955,3.7144,0.0000
C01057=21.543,108.678,52.574,179.2931,-1.6619,0.0000
C01058=23.225,112.648,53.599,177.9599,-4.2629,0.0000
C01059=25.324,116.233,54.111,176.7691,-3.4884,0.0000
C01060=29.146,118.641,54.383,177.4450,-0.9091,0.0000
C01061=34.236,119.458,54.605,178.3657,0.0207,0.0000
C01062=39.702,118.443,54.831,179.9236,0.0242,0.0000
C01063=45.138,116.556,54.980,179.9901,0.0038,0.0000
C01064=50.500,114.334,54.980,179.9903,0.0044,0.0000
C01065=55.679,111.826,54.831,179.9289,0.0369,0.0000
C01066=60.261,108.678,54.605,178.8296,1.1411,0.0000
C01067=63.283,104.502,54.383,178.8352,2.4492,0.0000
C01068=64.283,100.096,54.111,-179.8173,4.7459,0.0000
C01069=63.232,96.077,53.599,-178.4237,4.4541,0.0000
C01070=61.614,92.080,52.574,-179.3244,1.6749,0.0000
C01071=60.264,88.428,51.254,178.7172,-3.9710,0.0000
C01072=59.785,85.245,49.983,178.7116,-16.4611,0.0000
C01073=60.912,82.213,49.066,-160.4155,-30.4370,0.0000
C01074=64.361,78.707,48.701,-150.0629,-27.9242,0.0000
C01075=68.164,75.384,48.686,-149.5944,-27.7684,0.0000
C01076=71.867,71.867,48.696,-150.8705,-29.1299,0.0000
C01077=75.384,68.164,48.686,-152.2313,-30.4054,0.0000
C01078=78.707,64.361,48.701,-152.0749,-29.9360,0.0000
C01079=82.213,60.912,49.066,-149.5631,-19.5854,0.0000
C01080=85.245,59.785,49.983,-163.5389,1.2884,0.0000
C01081=88.428,60.264,51.254,-176.0290,1.2828,0.0000
C01082=92.080,61.614,52.574,178.3251,-0.6756,0.0000
C01083=96.077,63.232,53.599,175.5459,-1.5763,0.0000
C01084=100.096,64.283,54.111,175.2541,-0.1827,0.0000
C01085=104.502,63.283,54.383,177.5508,1.1648,0.0000
C01086=108.678,60.261,54.605,178.8589,1.1704,0.0000
C01087=111.826,55.679,54.831,179.9631,0.0711,0.0000
C01088=114.334,50.500,54.980,179.9956,0.0097,0.0000
C01089=116.556,45.138,54.980,179.9962,0.0099,0.0000
C01090=118.443,39.702,54.831,179.9758,0.0764,0.0000
C01091=119.458,34.236,54.605,179.9793,1.6343,0.0000
C01092=118.641,29.146,54.383,-179.0909,2.5550,0.0000
C01093=116.233,25.324,54.111,-176.5116,3.2309,0.0000
C01094=112.648,23.225,53.599,-175.7371,2.0401,0.0000
C01095=108.678,21.543,52.574,-178.3381,0.7069,0.0000
C01096=105.141,19.915,51.254,176.2856,-1.9045,0.0000
C01097=102.552,18.003,49.983,167.3286,-10.9254,0.0000
C01098=101.204,15.062,49.066,170.6921,-33.7051,0.0000
C01099=101.164,10.144,48.701,-178.1421,-38.0251,0.0000
C01100=101.503,5.105,48.686,-177.5588,-38.2122,0.0000
C01101=101.635,0.000,48.696,179.9997,-38.2417,0.0000
C01102=101.503,-5.105,48.686,177.5593,-38.2122,0.0000
C01103=101.164,-10.145,48.701,178.1439,-38.0249,0.0000
C01104=101.204,-15.062,49.066,-170.6930,-33.7055,0.0000
C01105=102.552,-18.003,49.983,-167.3286,-10.9254,0.0000
C01106=105.141,-19.915,51.254,-176.2856,-1.9045,0.0000
C01107=108.678,-21.543,52.574,178.3381,0.7069,0.0000
C01108=112.648,-23.225,53.599,175.7371,2.0401,0.0000
C01109=116.233,-25.324,54.111,176.5116,3.2309,0.0000
C01110=118.641,-29.146,54.383,179.0909,2.5550,0.0000
C01111=119.458,-34.236,54.605,-179.9793,1.6343,0.0000
C01112=118.443,-39.702,54.831,-179.9758,0.0764,0.0000
C01113=116.556,-45.138,54.980,-179.9962,0.0099,0.0000
C01114=114.334,-50.500,54.980,-179.9956,0.0097,0.0000
C01115=111.826,-55.679,54.831,-179.9631,0.0711,0.0000
C01116=108.678,-60.261,54.605,-178.8589,1.1704,0.0000
C01117=104.502,-63.283,54.383,-177.5508,1.1648,0.0000
C01118=100.096,-64.283,54.111,-175.2541,-0.1827,0.0000
C01119=96.077,-63.232,53.599,-175.5459,-1.5763,0.0000
C01120=92.080,-61.614,52.574,-178.3251,-0.6756,0.0000
C01121=88.428,-60.264,51.254,176.0290,1.2828,0.0000
C01122=85.245,-59.785,49.983,163.5389,1.2884,0.0000
C01123=82.213,-60.912,49.066,149.5630,-19.5845,0.0000
C01124=78.707,-64.361,48.701,152.0758,-29.9371,0.0000
C01125=75.384,-68.164,48.686,152.2316,-30.4056,0.0000
C01126=71.867,-71.867,48.696,150.8701,-29.1295,0.0000
C01127=68.164,-75.384,48.686,149.5946,-27.7687,0.0000
C01128=64.361,-78.707,48.701,150.0640,-27.9251,0.0000
C01129=60.912,-82.213,49.066,160.4146,-30.4369,0.0000
C01130=59.785,-85.245,49.983,-178.7116,-16.4611,0.0000
C01131=60.264,-88.428,51.254,-178.7172,-3.9710,0.0000
C01132=61.614,-92.080,52.574,179.3244,1.6749,0.0000
C01133=63.232,-96.077,53.599,178.4237,4.4541,0.0000
C01134=64.283,-100.096,54.111,179.8173,4.7459,0.0000
C01135=63.283,-104.502,54.383,-178.8352,2.4492,0.0000
C01136=60.261,-108.678,54.605,-178.8296,1.1411,0.0000
C01137=55.679,-111.826,54.831,-179.9289,0.0369,0.0000
C01138=50.500,-114.334,54.980,-179.9903,0.0044,0.0000
C01139=45.138,-116.556,54.980,-179.9901,0.0038,0.0000
C01140=39.702,-118.443,54.831,-179.9236,0.0242,0.0000
C01141=34.236,-119.458,54.605,-178.3657,0.0207,0.0000
C01142=29.146,-118.641,54.383,-177.4450,-0.9091,0.0000
C01143=25.324,-116.233,54.111,-176.7691,-3.4884,0.0000
C01144=23.225,-112.648,53.599,-177.9599,-4.2629,0.0000
C01145=21.543,-108.678,52.574,-179.2931,-1.6619,0.0000
C01146=19.915,-105.141,51.254,178.0955,3.7144,0.0000
C01147=18.003,-102.552,49.983,169.0746,12.6714,0.0000
C01148=15.062,-101.204,49.066,146.2949,9.3079,0.0000
C01149=10.144,-101.164,48.701,141.9749,-1.8579,0.0000
C01150=5.105,-101.503,48.686,141.7878,-2.4412,0.0000
C01151=0.000,-101.635,48.696,141.7583,0.0003,0.0000
C01152=0.000,-101.635,48.696,141.7583,0.0003,0.0000
C01153=-5.105,-101.503,48.686,141.7878,2.4407,0.0000
C01154=-10.145,-101.164,48.701,141.9751,1.8561,0.0000
C01155=-15.062,-101.204,49.066,146.2945,-9.3070,0.0000
C01156=-18.003,-102.552,49.983,169.0746,-12.6714,0.0000
C01157=-19.915,-105.141,51.254,178.0955,-3.7144,0.0000
C01158=-21.543,-108.678,52.574,-179.2931,1.6619,0.0000
C01159=-23.225,-112.648,53.599,-177.9599,4.2629,0.0000
C01160=-25.324,-116.233,54.111,-176.7691,3.4884,0.0000
C01161=-29.146,-118.641,54.383,-177.4450,0.9091,0.0000
C01162=-34.236,-119.458,54.605,-178.3657,-0.0207,0.0000
C01163=-39.702,-118.443,54.831,-179.9236,-0.0242,0.0000
C01164=-45.138,-116.556,54.980,-179.9901,-0.0038,0.0000
C01165=-50.500,-114.334,54.980,-179.9903,-0.0044,0.0000
C01166=-55.679,-111.826,54.831,-179.9289,-0.0369,0.0000
C01167=-60.261,-108.678,54.605,-178.8296,-1.1411,0.0000
C01168=-63.283,-104.502,54.383,-178.8352,-2.4492,0.0000
C01169=-64.283,-100.096,54.111,179.8173,-4.7459,0.0000
C01170=-63.232,-96.077,53.599,178.4237,-4.4541,0.0000
C01171=-61.614,-92.080,52.574,179.3244,-1.6749,0.0000
C01172=-60.264,-88.428,51.254,-178.7172,3.9710,0.0000
C01173=-59.785,-85.245,49.983,-178.7116,16.4611,0.0000
C01174=-60.912,-82.213,49.066,160.4155,30.4370,0.0000
C01175=-64.361,-78.707,48.701,150.0629,27.9242,0.0000
C01176=-68.164,-75.384,48.686,149.5944,27.7684,0.0000
C01177=-71.867,-71.867,48.696,150.8705,29.1299,0.0000
C01178=-75.384,-68.164,48.686,152.2313,30.4054,0.0000
C01179=-78.707,-64.361,48.701,152.0749,29.9360,0.0000
C01180=-82.213,-60.912,49.066,149.5631,19.5854,0.0000
C01181=-85.245,-59.785,49.983,163.5389,-1.2884,0.0000
C01182=-88.428,-60.264,51.254,176.0290,-1.2828,0.0000
C01183=-92.080,-61.614,52.574,-178.3251,0.6756,0.0000
C01184=-96.077,-63.232,53.599,-175.5459,1.5763,0.0000
C01185=-100.096,-64.283,54.111,-175.2541,0.1827,0.0000
C01186=-104.502,-63.283,54.383,-177.5508,-1.1648,0.0000
C01187=-108.678,-60.261,54.605,-178.8589,-1.1704,0.0000
C01188=-111.826,-55.679,54.831,-179.9631,-0.0711,0.0000
C01189=-114.334,-50.500,54.980,-179.9956,-0.0097,0.0000
C01190=-116.556,-45.138,54.980,-179.9962,-0.0099,0.0000
C01191=-118.443,-39.702,54.831,-179.9758,-0.0764,0.0000
C01192=-119.458,-34.236,54.605,-179.9793,-1.6343,0.0000
C01193=-118.641,-29.146,54.383,179.0909,-2.5550,0.0000
C01194=-116.233,-25.324,54.111,176.5116,-3.2309,0.0000
C01195=-112.648,-23.225,53.599,175.7371,-2.0401,0.0000
C01196=-108.678,-21.543,52.574,178.3381,-0.7069,0.0000
C01197=-105.141,-19.915,51.254,-176.2856,1.9045,0.0000
C01198=-102.552,-18.003,49.983,-167.3286,10.9254,0.0000
C01199=-101.204,-15.062,49.066,-170.6921,33.7051,0.0000
C01200=-101.164,-10.144,48.701,178.1421,38.0251,0.0000
C01201=-101.503,-5.105,48.686,177.5588,38.2122,0.0000
C01202=-101.635,0.000,48.696,-179.9997,38.2417,0.0000
C01203=-101.503,5.105,48.686,-177.5593,38.2122,0.0000
C01204=-101.164,10.145,48.701,-178.1439,38.0249,0.0000
C01205=-101.204,15.062,49.066,170.6930,33.7055,0.0000
C01206=-102.552,18.003,49.983,167.3286,10.9254,0.0000
C01207=-105.141,19.915,51.254,176.2856,1.9045,0.0000
C01208=-108.678,21.543,52.574,-178.3381,-0.7069,0.0000
C01209=-112.648,23.225,53.599,-175.7371,-2.0401,0.0000
C01210=-116.233,25.324,54.111,-176.5116,-3.2309,0.0000
C01211=-118.641,29.146,54.383,-179.0909,-2.5550,0.0000
C01212=-119.458,34.236,54.605,179.9793,-1.6343,0.0000
C01213=-118.443,39.702,54.831,179.9758,-0.0764,0.0000
C01214=-116.556,45.138,54.980,179.9962,-0.0099,0.0000
C01215=-114.334,50.500,54.980,179.9956,-0.0097,0.0000
C01216=-111.826,55.679,54.831,179.9631,-0.0711,0.0000
C01217=-108.678,60.261,54.605,178.8589,-1.1704,0.0000
C01218=-104.502,63.283,54.383,177.5508,-1.1648,0.0000
C01219=-100.096,64.283,54.111,175.2541,0.1827,0.0000
C01220=-96.077,63.232,53.599,175.5459,1.5763,0.0000
C01221=-92.080,61.614,52.574,178.3251,0.6756,0.0000
C01222=-88.428,60.264,51.254,-176.0290,-1.2828,0.0000
C01223=-85.245,59.785,49.983,-163.5389,-1.2884,0.0000
C01224=-82.213,60.912,49.066,-149.5630,19.5845,0.0000
C01225=-78.707,64.361,48.701,-152.0758,29.9371,0.0000
C01226=-75.384,68.164,48.686,-152.2316,30.4056,0.0000
C01227=-71.867,71.867,48.696,-150.8701,29.1295,0.0000
C01228=-68.164,75.384,48.686,-149.5946,27.7687,0.0000
C01229=-64.361,78.707,48.701,-150.0640,27.9251,0.0000
C01230=-60.912,82.213,49.066,-160.4146,30.4369,0.0000
C01231=-59.785,85.245,49.983,178.7116,16.4611,0.0000
C01232=-60.264,88.428,51.254,178.7172,3.9710,0.0000
C01233=-61.614,92.080,52.574,-179.3244,-1.6749,0.0000
C01234=-63.232,96.077,53.599,-178.4237,-4.4541,0.0000
C01235=-64.283,100.096,54.111,-179.8173,-4.7459,0.0000
C01236=-63.283,104.502,54.383,178.8352,-2.4492,0.0000
C01237=-60.261,108.678,54.605,178.8296,-1.1411,0.0000
C01238=-55.679,111.826,54.831,179.9289,-0.0369,0.0000
C01239=-50.500,114.334,54.980,179.9903,-0.0044,0.0000
C01240=-45.138,116.556,54.980,179.9901,-0.0038,0.0000
C01241=-39.702,118.443,54.831,179.9236,-0.0242,0.0000
C01242=-34.236,119.458,54.605,178.3657,-0.0207,0.0000
C01243=-29.146,118.641,54.383,177.4450,0.9091,0.0000
C01244=-25.324,116.233,54.111,176.7691,3.4884,0.0000
C01245=-23.225,112.648,53.599,177.9599,4.2629,0.0000
C01246=-21.543,108.678,52.574,179.2931,1.6619,0.0000
C01247=-19.915,105.141,51.254,-178.0955,-3.7144,0.0000
C01248=-18.003,102.552,49.983,-169.0746,-12.6714,0.0000
C01249=-15.062,101.204,49.066,-146.2945,-9.3070,0.0000
C01250=-10.145,101.164,48.701,-141.9751,1.8561,0.0000
C01251=-5.105,101.503,48.686,-141.7878,2.4407,0.0000
C01252=0.000,101.635,48.696,-141.7583,0.0003,0.0000
C01253=0.000,100.268,50.421,-141.4608,0.0003,0.0000
C01254=4.980,100.142,50.409,-141.4901,-2.4523,0.0000
C01255=9.934,99.815,50.426,-141.6887,-1.6526,0.0000
C01256=14.804,99.896,50.816,-146.5237,10.2391,0.0000
C01257=17.684,101.350,51.799,-170.4740,12.0658,0.0000
C01258=19.545,104.111,53.163,-178.6245,2.8992,0.0000
C01259=21.134,107.879,54.583,179.0883,-2.3066,0.0000
C01260=22.780,112.118,55.687,177.8524,-4.8646,0.0000
C01261=24.837,115.968,56.240,176.5275,-4.0634,0.0000
C01262=28.685,118.586,56.533,177.1534,-1.1005,0.0000
C01263=33.869,119.524,56.773,178.2332,-0.0001,0.0000
C01264=39.470,118.520,57.017,179.9127,0.0274,0.0000
C01265=45.059,116.586,57.178,179.9888,0.0042,0.0000
C01266=50.577,114.300,57.178,179.9891,0.0049,0.0000
C01267=55.897,111.716,57.017,179.9189,0.0423,0.0000
C01268=60.567,108.466,56.773,178.7506,1.2496,0.0000
C01269=63.569,104.136,56.533,178.7639,2.7906,0.0000
C01270=64.440,99.564,56.240,-179.5804,5.3211,0.0000
C01271=63.172,95.387,55.687,-178.0719,4.9550,0.0000
C01272=61.338,91.226,54.583,-179.0129,2.2754,0.0000
C01273=59.798,87.438,53.163,178.9211,-3.0218,0.0000
C01274=59.161,84.170,51.799,178.1391,-15.0993,0.0000
C01275=60.169,81.106,50.816,-161.2284,-30.7666,0.0000
C01276=63.555,77.604,50.426,-149.9263,-28.2920,0.0000
C01277=67.289,74.333,50.409,-149.3345,-28.0297,0.0000
C01278=70.900,70.900,50.421,-150.6099,-29.3905,0.0000
C01279=74.333,67.290,50.409,-151.9700,-30.6653,0.0000
C01280=77.605,63.555,50.426,-151.7071,-30.0725,0.0000
C01281=81.106,60.169,50.816,-149.2335,-18.7726,0.0000
C01282=84.170,59.161,51.799,-164.9007,1.8609,0.0000
C01283=87.438,59.798,53.163,-176.9782,1.0789,0.0000
C01284=91.226,61.338,54.583,177.7246,-0.9871,0.0000
C01285=95.387,63.172,55.687,175.0450,-1.9281,0.0000
C01286=99.564,64.440,56.240,174.6789,-0.4196,0.0000
C01287=104.136,63.569,56.533,177.2094,1.2361,0.0000
C01288=108.466,60.567,56.773,178.7504,1.2494,0.0000
C01289=111.716,55.897,57.017,179.9577,0.0811,0.0000
C01290=114.300,50.577,57.178,179.9951,0.0109,0.0000
C01291=116.586,45.059,57.178,179.9958,0.0112,0.0000
C01292=118.520,39.470,57.017,179.9726,0.0873,0.0000
C01293=119.524,33.869,56.773,-179.9999,1.7668,0.0000
C01294=118.586,28.685,56.533,-178.8995,2.8466,0.0000
C01295=115.968,24.837,56.240,-175.9366,3.4725,0.0000
C01296=112.118,22.780,55.687,-175.1354,2.1476,0.0000
C01297=107.879,21.134,54.583,-177.6934,0.9117,0.0000
C01298=104.111,19.545,53.163,177.1008,-1.3755,0.0000
C01299=101.350,17.684,51.799,167.9342,-9.5260,0.0000
C01300=99.896,14.804,50.816,169.7609,-33.4763,0.0000
C01301=99.815,9.934,50.426,-178.3474,-38.3113,0.0000
C01302=100.142,4.980,50.409,-177.5477,-38.5099,0.0000
C01303=100.268,0.000,50.421,179.9997,-38.5392,0.0000
C01304=100.142,-4.980,50.409,177.5481,-38.5100,0.0000
C01305=99.815,-9.935,50.426,178.3493,-38.3110,0.0000
C01306=99.896,-14.804,50.816,-169.7617,-33.4767,0.0000
C01307=101.350,-17.684,51.799,-167.9342,-9.5260,0.0000
C01308=104.111,-19.545,53.163,-177.1008,-1.3755,0.0000
C01309=107.879,-21.134,54.583,177.6934,0.9117,0.0000
C01310=112.118,-22.780,55.687,175.1354,2.1476,0.0000
C01311=115.968,-24.837,56.240,175.9366,3.4725,0.0000
C01312=118.586,-28.685,56.533,178.8995,2.8466,0.0000
C01313=119.524,-33.869,56.773,179.9999,1.7668,0.0000
C01314=118.520,-39.470,57.017,-179.9726,0.0873,0.0000
C01315=116.586,-45.059,57.178,-179.9958,0.0112,0.0000
C01316=114.300,-50.577,57.178,-179.9951,0.0109,0.0000
C01317=111.716,-55.897,57.017,-179.9577,0.0811,0.0000
C01318=108.466,-60.567,56.773,-178.7504,1.2494,0.0000
C01319=104.136,-63.569,56.533,-177.2094,1.2361,0.0000
C01320=99.564,-64.440,56.240,-174.6789,-0.4196,0.0000
C01321=95.387,-63.172,55.687,-175.0450,-1.9281,0.0000
C01322=91.226,-61.338,54.583,-177.7246,-0.9871,0.0000
C01323=87.438,-59.798,53.163,176.9782,1.0789,0.0000
C01324=84.170,-59.161,51.799,164.9007,1.8609,0.0000
C01325=81.106,-60.169,50.816,149.2334,-18.7716,0.0000
C01326=77.604,-63.555,50.426,151.7080,-30.0737,0.0000
C01327=74.333,-67.289,50.409,151.9703,-30.6655,0.0000
C01328=70.900,-70.900,50.421,150.6095,-29.3901,0.0000
C01329=67.290,-74.333,50.409,149.3347,-28.0300,0.0000
C01330=63.555,-77.605,50.426,149.9275,-28.2929,0.0000
C01331=60.169,-81.106,50.816,161.2274,-30.7665,0.0000
C01332=59.161,-84.170,51.799,-178.1391,-15.0993,0.0000
C01333=59.798,-87.438,53.163,-178.9211,-3.0218,0.0000
C01334=61.338,-91.226,54.583,179.0129,2.2754,0.0000
C01335=63.172,-95.387,55.687,178.0719,4.9550,0.0000
C01336=64.440,-99.564,56.240,179.5804,5.3211,0.0000
C01337=63.569,-104.136,56.533,-178.7639,2.7906,0.0000
C01338=60.567,-108.466,56.773,-178.7506,1.2496,0.0000
C01339=55.897,-111.716,57.017,-179.9189,0.0423,0.0000
C01340=50.577,-114.300,57.178,-179.9891,0.0049,0.0000
C01341=45.059,-116.586,57.178,-179.9888,0.0042,0.0000
C01342=39.470,-118.520,57.017,-179.9127,0.0274,0.0000
C01343=33.869,-119.524,56.773,-178.2332,-0.0001,0.0000
C01344=28.685,-118.586,56.533,-177.1534,-1.1005,0.0000
C01345=24.837,-115.968,56.240,-176.5275,-4.0634,0.0000
C01346=22.780,-112.118,55.687,-177.8524,-4.8646,0.0000
C01347=21.134,-107.879,54.583,-179.0883,-2.3066,0.0000
C01348=19.545,-104.111,53.163,178.6245,2.8992,0.0000
C01349=17.684,-101.350,51.799,170.4740,12.0658,0.0000
C01350=14.804,-99.896,50.816,146.5237,10.2391,0.0000
C01351=9.934,-99.815,50.426,141.6887,-1.6526,0.0000
C01352=4.980,-100.142,50.409,141.4901,-2.4523,0.0000
C01353=0.000,-100.268,50.421,141.4608,0.0003,0.0000
C01354=0.000,-100.268,50.421,141.4608,0.0003,0.0000
C01355=-4.980,-100.142,50.409,141.4900,2.4519,0.0000
C01356=-9.935,-99.815,50.426,141.6890,1.6507,0.0000
C01357=-14.804,-99.896,50.816,146.5233,-10.2383,0.0000
C01358=-17.684,-101.350,51.799,170.4740,-12.0658,0.0000
C01359=-19.545,-104.111,53.163,178.6245,-2.8992,0.0000
C01360=-21.134,-107.879,54.583,-179.0883,2.3066,0.0000
C01361=-22.780,-112.118,55.687,-177.8524,4.8646,0.0000
C01362=-24.837,-115.968,56.240,-176.5275,4.0634,0.0000
C01363=-28.685,-118.586,56.533,-177.1534,1.1005,0.0000
C01364=-33.869,-119.524,56.773,-178.2332,0.0001,0.0000
C01365=-39.470,-118.520,57.017,-179.9127,-0.0274,0.0000
C01366=-45.059,-116.586,57.178,-179.9888,-0.0042,0.0000
C01367=-50.577,-114.300,57.178,-179.9891,-0.0049,0.0000
C01368=-55.897,-111.716,57.017,-179.9189,-0.0423,0.0000
C01369=-60.567,-108.466,56.773,-178.7506,-1.2496,0.0000
C01370=-63.569,-104.136,56.533,-178.7639,-2.7906,0.0000
C01371=-64.440,-99.564,56.240,179.5804,-5.3211,0.0000
C01372=-63.172,-95.387,55.687,178.0719,-4.9550,0.0000
C01373=-61.338,-91.226,54.583,179.0129,-2.2754,0.0000
C01374=-59.798,-87.438,53.163,-178.9211,3.0218,0.0000
C01375=-59.161,-84.170,51.799,-178.1391,15.0993,0.0000
C01376=-60.169,-81.106,50.816,161.2284,30.7666,0.0000
C01377=-63.555,-77.604,50.426,149.9263,28.2920,0.0000
C01378=-67.289,-74.333,50.409,149.3345,28.0297,0.0000
C01379=-70.900,-70.900,50.421,150.6099,29.3905,0.0000
C01380=-74.333,-67.290,50.409,151.9700,30.6653,0.0000
C01381=-77.605,-63.555,50.426,151.7071,30.0725,0.0000
C01382=-81.106,-60.169,50.816,149.2335,18.7726,0.0000
C01383=-84.170,-59.161,51.799,164.9007,-1.8609,0.0000
C01384=-87.438,-59.798,53.163,176.9782,-1.0789,0.0000
C01385=-91.226,-61.338,54.583,-177.7246,0.9871,0.0000
C01386=-95.387,-63.172,55.687,-175.0450,1.9281,0.0000
C01387=-99.564,-64.440,56.240,-174.6789,0.4196,0.0000
C01388=-104.136,-63.569,56.533,-177.2094,-1.2361,0.0000
C01389=-108.466,-60.567,56.773,-178.7504,-1.2494,0.0000
C01390=-111.716,-55.897,57.017,-179.9577,-0.0811,0.0000
C01391=-114.300,-50.577,57.178,-179.9951,-0.0109,0.0000
C01392=-116.586,-45.059,57.178,-179.9958,-0.0112,0.0000
C01393=-118.520,-39.470,57.017,-179.9726,-0.0873,0.0000
C01394=-119.524,-33.869,56.773,179.9999,-1.7668,0.0000
C01395=-118.586,-28.685,56.533,178.8995,-2.8466,0.0000
C01396=-115.968,-24.837,56.240,175.9366,-3.4725,0.0000
C01397=-112.118,-22.780,55.687,175.1354,-2.1476,0.0000
C01398=-107.879,-21.134,54.583,177.6934,-0.9117,0.0000
C01399=-104.111,-19.545,53.163,-177.1008,1.3755,0.0000
C01400=-101.350,-17.684,51.799,-167.9342,9.5260,0.0000
C01401=-99.896,-14.804,50.816,-169.7609,33.4763,0.0000
C01402=-99.815,-9.934,50.426,178.3474,38.3113,0.0000
C01403=-100.142,-4.980,50.409,177.5477,38.5099,0.0000
C01404=-100.268,0.000,50.421,-179.9997,38.5392,0.0000
C01405=-100.142,4.980,50.409,-177.5481,38.5100,0.0000
C01406=-99.815,9.935,50.426,-178.3493,38.3110,0.0000
C01407=-99.896,14.804,50.816,169.7617,33.4767,0.0000
C01408=-101.350,17.684,51.799,167.9342,9.5260,0.0000
C01409=-104.111,19.545,53.163,177.1008,1.3755,0.0000
C01410=-107.879,21.134,54.583,-177.6934,-0.9117,0.0000
C01411=-112.118,22.780,55.687,-175.1354,-2.1476,0.0000
C01412=-115.968,24.837,56.240,-175.9366,-3.4725,0.0000
C01413=-118.586,28.685,56.533,-178.8995,-2.8466,0.0000
C01414=-119.524,33.869,56.773,-179.9999,-1.7668,0.0000
C01415=-118.520,39.470,57.017,179.9726,-0.0873,0.0000
C01416=-116.586,45.059,57.178,179.9958,-0.0112,0.0000
C01417=-114.300,50.577,57.178,179.9951,-0.0109,0.0000
C01418=-111.716,55.897,57.017,179.9577,-0.0811,0.0000
C01419=-108.466,60.567,56.773,178.7504,-1.2494,0.0000
C01420=-104.136,63.569,56.533,177.2094,-1.2361,0.0000
C01421=-99.564,64.440,56.240,174.6789,0.4196,0.0000
C01422=-95.387,63.172,55.687,175.0450,1.9281,0.0000
C01423=-91.226,61.338,54.583,177.7246,0.9871,0.0000
C01424=-87.438,59.798,53.163,-176.9782,-1.0789,0.0000
C01425=-84.170,59.161,51.799,-164.9007,-1.8609,0.0000
C01426=-81.106,60.169,50.816,-149.2334,18.7716,0.0000
C01427=-77.604,63.555,50.426,-151.7080,30.0737,0.0000
C01428=-74.333,67.289,50.409,-151.9703,30.6655,0.0000
C01429=-70.900,70.900,50.421,-150.6095,29.3901,0.0000
C01430=-67.290,74.333,50.409,-149.3347,28.0300,0.0000
C01431=-63.555,77.605,50.426,-149.9275,28.2929,0.0000
C01432=-60.169,81.106,50.816,-161.2274,30.7665,0.0000
C01433=-59.161,84.170,51.799,178.1391,15.0993,0.0000
C01434=-59.798,87.438,53.163,178.9211,3.0218,0.0000
C01435=-61.338,91.226,54.583,-179.0129,-2.2754,0.0000
C01436=-63.172,95.387,55.687,-178.0719,-4.9550,0.0000
C01437=-64.440,99.564,56.240,-179.5804,-5.3211,0.0000
C01438=-63.569,104.136,56.533,178.7639,-2.7906,0.0000
C01439=-60.567,108.466,56.773,178.7506,-1.2496,0.0000
C01440=-55.897,111.716,57.017,179.9189,-0.0423,0.0000
C01441=-50.577,114.300,57.178,179.9891,-0.0049,0.0000
C01442=-45.059,116.586,57.178,179.9888,-0.0042,0.0000
C01443=-39.470,118.520,57.017,179.9127,-0.0274,0.0000
C01444=-33.869,119.524,56.773,178.2332,0.0001,0.0000
C01445=-28.685,118.586,56.533,177.1534,1.1005,0.0000
C01446=-24.837,115.968,56.240,176.5275,4.0634,0.0000
C01447=-22.780,112.118,55.687,177.8524,4.8646,0.0000
C01448=-21.134,107.879,54.583,179.0883,2.3066,0.0000
C01449=-19.545,104.111,53.163,-178.6245,-2.8992,0.0000
C01450=-17.684,101.350,51.799,-170.4740,-12.0658,0.0000
C01451=-14.804,99.896,50.816,-146.5233,-10.2383,0.0000
C01452=-9.935,99.815,50.426,-141.6890,1.6507,0.0000
C01453=-4.980,100.142,50.409,-141.4900,2.4519,0.0000
C01454=0.000,100.268,50.421,-141.4608,0.0003,0.0000
C01455=0.000,98.894,52.138,-141.2150,0.0003,0.0000
C01456=4.855,98.772,52.126,-141.2439,-2.4580,0.0000
C01457=9.723,98.457,52.144,-141.4560,-1.4330,0.0000
C01458=14.545,98.581,52.560,-146.8469,11.1315,0.0000
C01459=17.363,100.142,53.609,-171.7702,11.3500,0.0000
C01460=19.173,103.076,55.068,-179.0687,2.1138,0.0000
C01461=20.723,107.076,56.590,178.9313,-2.8990,0.0000
C01462=22.333,111.586,57.775,177.7894,-5.4074,0.0000
C01463=24.347,115.701,58.368,176.3498,-4.6056,0.0000
C01464=28.222,118.530,58.683,176.8892,-1.2960,0.0000
C01465=33.501,119.591,58.941,178.1098,-0.0233,0.0000
C01466=39.236,118.597,59.203,179.9025,0.0305,0.0000
C01467=44.979,116.617,59.377,179.9877,0.0047,0.0000
C01468=50.655,114.266,59.377,179.9880,0.0054,0.0000
C01469=56.117,111.605,59.203,179.9095,0.0474,0.0000
C01470=60.875,108.253,58.941,178.6797,1.3533,0.0000
C01471=63.857,103.770,58.683,178.7149,3.1153,0.0000
C01472=64.597,99.029,58.368,-179.3209,5.8281,0.0000
C01473=63.112,94.695,57.775,-177.7301,5.3830,0.0000
C01474=61.061,90.368,56.590,-178.7043,2.8052,0.0000
C01475=59.329,86.443,55.068,179.1633,-2.1530,0.0000
C01476=58.533,83.089,53.609,177.7286,-13.7234,0.0000
C01477=59.422,79.992,52.560,-162.1120,-31.0069,0.0000
C01478=62.744,76.495,52.144,-149.8419,-28.6194,0.0000
C01479=66.410,73.275,52.126,-149.1210,-28.2484,0.0000
C01480=69.928,69.928,52.138,-150.3939,-29.6064,0.0000
C01481=73.275,66.410,52.126,-151.7514,-30.8788,0.0000
C01482=76.495,62.744,52.144,-151.3797,-30.1568,0.0000
C01483=79.992,59.422,52.560,-148.9931,-17.8889,0.0000
C01484=83.089,58.533,53.609,-166.2766,2.2714,0.0000
C01485=86.443,59.329,55.068,-177.8470,0.8367,0.0000
C01486=90.368,61.061,56.590,177.1948,-1.2957,0.0000
C01487=94.695,63.112,57.775,174.6170,-2.2699,0.0000
C01488=99.029,64.597,58.368,174.1719,-0.6791,0.0000
C01489=103.770,63.857,58.683,176.8847,1.2851,0.0000
C01490=108.253,60.875,58.941,178.6467,1.3203,0.0000
C01491=111.605,56.117,59.203,179.9526,0.0905,0.0000
C01492=114.266,50.655,59.377,179.9946,0.0120,0.0000
C01493=116.617,44.979,59.377,179.9953,0.0123,0.0000
C01494=118.597,39.236,59.203,179.9695,0.0975,0.0000
C01495=119.591,33.501,58.941,-179.9767,1.8902,0.0000
C01496=118.530,28.222,58.683,-178.7040,3.1108,0.0000
C01497=115.701,24.347,58.368,-175.3944,3.6502,0.0000
C01498=111.586,22.333,57.775,-174.5926,2.2106,0.0000
C01499=107.076,20.723,56.590,-177.1010,1.0687,0.0000
C01500=103.076,19.173,55.068,177.8862,-0.9313,0.0000
C01501=100.142,17.363,53.609,168.6500,-8.2298,0.0000
C01502=98.581,14.545,52.560,168.8685,-33.1531,0.0000
C01503=98.457,9.723,52.144,-178.5670,-38.5440,0.0000
C01504=98.772,4.855,52.126,-177.5420,-38.7561,0.0000
C01505=98.894,0.000,52.138,179.9997,-38.7850,0.0000
C01506=98.772,-4.855,52.126,177.5424,-38.7561,0.0000
C01507=98.457,-9.723,52.144,178.5690,-38.5438,0.0000
C01508=98.581,-14.545,52.560,-168.8693,-33.1536,0.0000
C01509=100.142,-17.363,53.609,-168.6500,-8.2298,0.0000
C01510=103.076,-19.173,55.068,-177.8862,-0.9313,0.0000
C01511=107.076,-20.723,56.590,177.1010,1.0687,0.0000
C01512=111.586,-22.333,57.775,174.5926,2.2106,0.0000
C01513=115.701,-24.347,58.368,175.3944,3.6502,0.0000
C01514=118.530,-28.222,58.683,178.7040,3.1108,0.0000
C01515=119.591,-33.501,58.941,179.9767,1.8902,0.0000
C01516=118.597,-39.236,59.203,-179.9695,0.0975,0.0000
C01517=116.617,-44.979,59.377,-179.9953,0.0123,0.0000
C01518=114.266,-50.655,59.377,-179.9946,0.0120,0.0000
C01519=111.605,-56.117,59.203,-179.9526,0.0905,0.0000
C01520=108.253,-60.875,58.941,-178.6467,1.3203,0.0000
C01521=103.770,-63.857,58.683,-176.8847,1.2851,0.0000
C01522=99.029,-64.597,58.368,-174.1719,-0.6791,0.0000
C01523=94.695,-63.112,57.775,-174.6170,-2.2699,0.0000
C01524=90.368,-61.061,56.590,-177.1948,-1.2957,0.0000
C01525=86.443,-59.329,55.068,177.8470,0.8367,0.0000
C01526=83.089,-58.533,53.609,166.2766,2.2714,0.0000
C01527=79.992,-59.422,52.560,148.9931,-17.8880,0.0000
C01528=76.495,-62.744,52.144,151.3806,-30.1581,0.0000
C01529=73.275,-66.410,52.126,151.7516,-30.8790,0.0000
C01530=69.928,-69.928,52.138,150.3936,-29.6061,0.0000
C01531=66.410,-73.275,52.126,149.1212,-28.2486,0.0000
C01532=62.744,-76.495,52.144,149.8432,-28.6203,0.0000
C01533=59.422,-79.992,52.560,162.1111,-31.0069,0.0000
C01534=58.533,-83.089,53.609,-177.7286,-13.7234,0.0000
C01535=59.329,-86.443,55.068,-179.1633,-2.1530,0.0000
C01536=61.061,-90.368,56.590,178.7043,2.8052,0.0000
C01537=63.112,-94.695,57.775,177.7301,5.3830,0.0000
C01538=64.597,-99.029,58.368,179.3209,5.8281,0.0000
C01539=63.857,-103.770,58.683,-178.7149,3.1153,0.0000
C01540=60.875,-108.253,58.941,-178.6797,1.3533,0.0000
C01541=56.117,-111.605,59.203,-179.9095,0.0474,0.0000
C01542=50.655,-114.266,59.377,-179.9880,0.0054,0.0000
C01543=44.979,-116.617,59.377,-179.9877,0.0047,0.0000
C01544=39.236,-118.597,59.203,-179.9025,0.0305,0.0000
C01545=33.501,-119.591,58.941,-178.1098,-0.0233,0.0000
C01546=28.222,-118.530,58.683,-176.8892,-1.2960,0.0000
C01547=24.347,-115.701,58.368,-176.3498,-4.6056,0.0000
C01548=22.333,-111.586,57.775,-177.7894,-5.4074,0.0000
C01549=20.723,-107.076,56.590,-178.9313,-2.8990,0.0000
C01550=19.173,-103.076,55.068,179.0687,2.1138,0.0000
C01551=17.363,-100.142,53.609,171.7702,11.3500,0.0000
C01552=14.545,-98.581,52.560,146.8469,11.1315,0.0000
C01553=9.723,-98.457,52.144,141.4560,-1.4330,0.0000
C01554=4.855,-98.772,52.126,141.2439,-2.4580,0.0000
C01555=0.000,-98.894,52.138,141.2150,0.0003,0.0000
C01556=0.000,-98.894,52.138,141.2150,0.0003,0.0000
C01557=-4.855,-98.772,52.126,141.2439,2.4576,0.0000
C01558=-9.723,-98.457,52.144,141.4562,1.4310,0.0000
C01559=-14.545,-98.581,52.560,146.8464,-11.1307,0.0000
C01560=-17.363,-100.142,53.609,171.7702,-11.3500,0.0000
C01561=-19.173,-103.076,55.068,179.0687,-2.1138,0.0000
C01562=-20.723,-107.076,56.590,-178.9313,2.8990,0.0000
C01563=-22.333,-111.586,57.775,-177.7894,5.4074,0.0000
C01564=-24.347,-115.701,58.368,-176.3498,4.6056,0.0000
C01565=-28.222,-118.530,58.683,-176.8892,1.2960,0.0000
C01566=-33.501,-119.591,58.941,-178.1098,0.0233,0.0000
C01567=-39.236,-118.597,59.203,-179.9025,-0.0305,0.0000
C01568=-44.979,-116.617,59.377,-179.9877,-0.0047,0.0000
C01569=-50.655,-114.266,59.377,-179.9880,-0.0054,0.0000
C01570=-56.117,-111.605,59.203,-179.9095,-0.0474,0.0000
C01571=-60.875,-108.253,58.941,-178.6797,-1.3533,0.0000
C01572=-63.857,-103.770,58.683,-178.7149,-3.1153,0.0000
C01573=-64.597,-99.029,58.368,179.3209,-5.8281,0.0000
C01574=-63.112,-94.695,57.775,177.7301,-5.3830,0.0000
C01575=-61.061,-90.368,56.590,178.7043,-2.8052,0.0000
C01576=-59.329,-86.443,55.068,-179.1633,2.1530,0.0000
C01577=-58.533,-83.089,53.609,-177.7286,13.7234,0.0000
C01578=-59.422,-79.992,52.560,162.1120,31.0069,0.0000
C01579=-62.744,-76.495,52.144,149.8419,28.6194,0.0000
C01580=-66.410,-73.275,52.126,149.1210,28.2484,0.0000
C01581=-69.928,-69.928,52.138,150.3939,29.6064,0.0000
C01582=-73.275,-66.410,52.126,151.7514,30.8788,0.0000
C01583=-76.495,-62.744,52.144,151.3797,30.1568,0.0000
C01584=-79.992,-59.422,52.560,148.9931,17.8889,0.0000
C01585=-83.089,-58.533,53.609,166.2766,-2.2714,0.0000
C01586=-86.443,-59.329,55.068,177.8470,-0.8367,0.0000
C01587=-90.368,-61.061,56.590,-177.1948,1.2957,0.0000
C01588=-94.695,-63.112,57.775,-174.6170,2.2699,0.0000
C01589=-99.029,-64.597,58.368,-174.1719,0.6791,0.0000
C01590=-103.770,-63.857,58.683,-176.8847,-1.2851,0.0000
C01591=-108.253,-60.875,58.941,-178.6467,-1.3203,0.0000
C01592=-111.605,-56.117,59.203,-179.9526,-0.0905,0.0000
C01593=-114.266,-50.655,59.377,-179.9946,-0.0120,0.0000
C01594=-116.617,-44.979,59.377,-179.9953,-0.0123,0.0000
C01595=-118.597,-39.236,59.203,-179.9695,-0.0975,0.0000
C01596=-119.591,-33.501,58.941,179.9767,-1.8902,0.0000
C01597=-118.530,-28.222,58.683,178.7040,-3.1108,0.0000
C01598=-115.701,-24.347,58.368,175.3944,-3.6502,0.0000
C01599=-111.586,-22.333,57.775,174.5926,-2.2106,0.0000
C01600=-107.076,-20.723,56.590,177.1010,-1.0687,0.0000
C01601=-103.076,-19.173,55.068,-177.8862,0.9313,0.0000
C01602=-100.142,-17.363,53.609,-168.6500,8.2298,0.0000
C01603=-98.581,-14.545,52.560,-168.8685,33.1531,0.0000
C01604=-98.457,-9.723,52.144,178.5670,38.5440,0.0000
C01605=-98.772,-4.855,52.126,177.5420,38.7561,0.0000
C01606=-98.894,0.000,52.138,-179.9997,38.7850,0.0000
C01607=-98.772,4.855,52.126,-177.5424,38.7561,0.0000
C01608=-98.457,9.723,52.144,-178.5690,38.5438,0.0000
C01609=-98.581,14.545,52.560,168.8693,33.1536,0.0000
C01610=-100.142,17.363,53.609,168.6500,8.2298,0.0000
C01611=-103.076,19.173,55.068,177.8862,0.9313,0.0000
C01612=-107.076,20.723,56.590,-177.1010,-1.0687,0.0000
C01613=-111.586,22.333,57.775,-174.5926,-2.2106,0.0000
C01614=-115.701,24.347,58.368,-175.3944,-3.6502,0.0000
C01615=-118.530,28.222,58.683,-178.7040,-3.1108,0.0000
C01616=-119.591,33.501,58.941,-179.9767,-1.8902,0.0000
C01617=-118.597,39.236,59.203,179.9695,-0.0975,0.0000
C01618=-116.617,44.979,59.377,179.9953,-0.0123,0.0000
C01619=-114.266,50.655,59.377,179.9946,-0.0120,0.0000
C01620=-111.605,56.117,59.203,179.9526,-0.0905,0.0000
C01621=-108.253,60.875,58.941,178.6467,-1.3203,0.0000
C01622=-103.770,63.857,58.683,176.8847,-1.2851,0.0000
C01623=-99.029,64.597,58.368,174.1719,0.6791,0.0000
C01624=-94.695,63.112,57.775,174.6170,2.2699,0.0000
C01625=-90.368,61.061,56.590,177.1948,1.2957,0.0000
C01626=-86.443,59.329,55.068,-177.8470,-0.8367,0.0000
C01627=-83.089,58.533,53.609,-166.2766,-2.2714,0.0000
C01628=-79.992,59.422,52.560,-148.9931,17.8880,0.0000
C01629=-76.495,62.744,52.144,-151.3806,30.1581,0.0000
C01630=-73.275,66.410,52.126,-151.7516,30.8790,0.0000
C01631=-69.928,69.928,52.138,-150.3936,29.6061,0.0000
C01632=-66.410,73.275,52.126,-149.1212,28.2486,0.0000
C01633=-62.744,76.495,52.144,-149.8432,28.6203,0.0000
C01634=-59.422,79.992,52.560,-162.1111,31.0069,0.0000
C01635=-58.533,83.089,53.609,177.7286,13.7234,0.0000
C01636=-59.329,86.443,55.068,179.1633,2.1530,0.0000
C01637=-61.061,90.368,56.590,-178.7043,-2.8052,0.0000
C01638=-63.112,94.695,57.775,-177.7301,-5.3830,0.0000
C01639=-64.597,99.029,58.368,-179.3209,-5.8281,0.0000
C01640=-63.857,103.770,58.683,178.7149,-3.1153,0.0000
C01641=-60.875,108.253,58.941,178.6797,-1.3533,0.0000
C01642=-56.117,111.605,59.203,179.9095,-0.0474,0.0000
C01643=-50.655,114.266,59.377,179.9880,-0.0054,0.0000
C01644=-44.979,116.617,59.377,179.9877,-0.0047,0.0000
C01645=-39.236,118.597,59.203,179.9025,-0.0305,0.0000
C01646=-33.501,119.591,58.941,178.1098,0.0233,0.0000
C01647=-28.222,118.530,58.683,176.8892,1.2960,0.0000
C01648=-24.347,115.701,58.368,176.3498,4.6056,0.0000
C01649=-22.333,111.586,57.775,177.7894,5.4074,0.0000
C01650=-20.723,107.076,56.590,178.9313,2.8990,0.0000
C01651=-19.173,103.076,55.068,-179.0687,-2.1138,0.0000
C01652=-17.363,100.142,53.609,-171.7702,-11.3500,0.0000
C01653=-14.545,98.581,52.560,-146.8464,-11.1307,0.0000
C01654=-9.723,98.457,52.144,-141.4562,1.4310,0.0000
C01655=-4.855,98.772,52.126,-141.2439,2.4576,0.0000
C01656=0.000,98.894,52.138,-141.2150,0.0003,0.0000
C01657=0.000,97.513,53.851,-141.0193,0.0002,0.0000
C01658=4.729,97.396,53.838,-141.0478,-2.4582,0.0000
C01659=9.511,97.093,53.857,-141.2751,-1.2004,0.0000
C01660=14.284,97.259,54.299,-147.2615,11.9753,0.0000
C01661=17.042,98.929,55.416,-172.9538,10.5519,0.0000
C01662=18.799,102.037,56.970,-179.4391,1.3661,0.0000
C01663=20.311,106.271,58.595,178.8138,-3.4384,0.0000
C01664=21.884,111.053,59.862,177.7620,-5.8906,0.0000
C01665=23.856,115.434,60.496,176.2287,-5.1072,0.0000
C01666=27.759,118.474,60.833,176.6541,-1.4916,0.0000
C01667=33.133,119.658,61.109,177.9965,-0.0483,0.0000
C01668=39.003,118.674,61.389,179.8930,0.0333,0.0000
C01669=44.900,116.647,61.575,179.9867,0.0050,0.0000
C01670=50.733,114.231,61.575,179.9870,0.0059,0.0000
C01671=56.336,111.494,61.389,179.9008,0.0521,0.0000
C01672=61.183,108.040,61.109,178.6171,1.4511,0.0000
C01673=64.145,103.402,60.833,178.6866,3.4195,0.0000
C01674=64.755,98.493,60.496,-179.0498,6.2664,0.0000
C01675=63.051,94.001,59.862,-177.4051,5.7440,0.0000
C01676=60.783,89.507,58.595,-178.4051,3.2696,0.0000
C01677=58.858,85.443,56.970,179.4304,-1.3626,0.0000
C01678=57.903,82.003,55.416,177.4625,-12.3592,0.0000
C01679=58.672,78.873,54.299,-163.0569,-31.1575,0.0000
C01680=61.930,75.380,53.857,-149.8083,-28.9069,0.0000
C01681=65.526,72.213,53.838,-148.9527,-28.4254,0.0000
C01682=68.952,68.952,53.851,-150.2215,-29.7787,0.0000
C01683=72.213,65.526,53.838,-151.5744,-31.0471,0.0000
C01684=75.380,61.930,53.857,-151.0921,-30.1904,0.0000
C01685=78.873,58.672,54.299,-148.8426,-16.9440,0.0000
C01686=82.003,57.903,55.416,-167.6408,2.5375,0.0000
C01687=85.443,58.858,56.970,-178.6374,0.5696,0.0000
C01688=89.507,60.783,58.595,176.7304,-1.5949,0.0000
C01689=94.001,63.051,59.862,174.2560,-2.5949,0.0000
C01690=98.493,64.755,60.496,173.7336,-0.9502,0.0000
C01691=103.402,64.145,60.833,176.5805,1.3134,0.0000
C01692=108.040,61.183,61.109,178.5489,1.3829,0.0000
C01693=111.494,56.336,61.389,179.9479,0.0992,0.0000
C01694=114.231,50.733,61.575,179.9941,0.0130,0.0000
C01695=116.647,44.900,61.575,179.9950,0.0133,0.0000
C01696=118.674,39.003,61.389,179.9667,0.1070,0.0000
C01697=119.658,33.133,61.109,-179.9517,2.0035,0.0000
C01698=118.474,27.759,60.833,-178.5084,3.3459,0.0000
C01699=115.434,23.856,60.496,-174.8928,3.7713,0.0000
C01700=111.053,21.884,59.862,-174.1094,2.2380,0.0000
C01701=106.271,20.311,58.595,-176.5616,1.1862,0.0000
C01702=102.037,18.799,56.970,178.6339,-0.5609,0.0000
C01703=98.929,17.042,55.416,169.4481,-7.0462,0.0000
C01704=97.259,14.284,54.299,168.0247,-32.7385,0.0000
C01705=97.093,9.511,53.857,-178.7996,-38.7249,0.0000
C01706=97.396,4.729,53.838,-177.5418,-38.9522,0.0000
C01707=97.513,0.000,53.851,179.9998,-38.9807,0.0000
C01708=97.396,-4.728,53.838,177.5421,-38.9522,0.0000
C01709=97.093,-9.511,53.857,178.8017,-38.7247,0.0000
C01710=97.259,-14.284,54.299,-168.0255,-32.7390,0.0000
C01711=98.929,-17.042,55.416,-169.4481,-7.0462,0.0000
C01712=102.037,-18.799,56.970,-178.6339,-0.5609,0.0000
C01713=106.271,-20.311,58.595,176.5616,1.1862,0.0000
C01714=111.053,-21.884,59.862,174.1094,2.2380,0.0000
C01715=115.434,-23.856,60.496,174.8928,3.7713,0.0000
C01716=118.474,-27.759,60.833,178.5084,3.3459,0.0000
C01717=119.658,-33.133,61.109,179.9517,2.0035,0.0000
C01718=118.674,-39.003,61.389,-179.9667,0.1070,0.0000
C01719=116.647,-44.900,61.575,-179.9950,0.0133,0.0000
C01720=114.231,-50.733,61.575,-179.9941,0.0130,0.0000
C01721=111.494,-56.336,61.389,-179.9479,0.0992,0.0000
C01722=108.040,-61.183,61.109,-178.5489,1.3829,0.0000
C01723=103.402,-64.145,60.833,-176.5805,1.3134,0.0000
C01724=98.493,-64.755,60.496,-173.7336,-0.9502,0.0000
C01725=94.001,-63.051,59.862,-174.2560,-2.5949,0.0000
C01726=89.507,-60.783,58.595,-176.7304,-1.5949,0.0000
C01727=85.443,-58.858,56.970,178.6374,0.5696,0.0000
C01728=82.003,-57.903,55.416,167.6408,2.5375,0.0000
C01729=78.873,-58.672,54.299,148.8425,-16.9431,0.0000
C01730=75.380,-61.930,53.857,151.0931,-30.1917,0.0000
C01731=72.213,-65.526,53.838,151.5746,-31.0473,0.0000
C01732=68.952,-68.952,53.851,150.2213,-29.7785,0.0000
C01733=65.526,-72.213,53.838,148.9529,-28.4256,0.0000
C01734=61.930,-75.380,53.857,149.8096,-28.9079,0.0000
C01735=58.672,-78.873,54.299,163.0560,-31.1574,0.0000
C01736=57.903,-82.003,55.416,-177.4625,-12.3592,0.0000
C01737=58.858,-85.443,56.970,-179.4304,-1.3626,0.0000
C01738=60.783,-89.507,58.595,178.4051,3.2696,0.0000
C01739=63.051,-94.001,59.862,177.4051,5.7440,0.0000
C01740=64.755,-98.493,60.496,179.0498,6.2664,0.0000
C01741=64.145,-103.402,60.833,-178.6866,3.4195,0.0000
C01742=61.183,-108.040,61.109,-178.6171,1.4511,0.0000
C01743=56.336,-111.494,61.389,-179.9008,0.0521,0.0000
C01744=50.733,-114.231,61.575,-179.9870,0.0059,0.0000
C01745=44.900,-116.647,61.575,-179.9867,0.0050,0.0000
C01746=39.003,-118.674,61.389,-179.8930,0.0333,0.0000
C01747=33.133,-119.658,61.109,-177.9965,-0.0483,0.0000
C01748=27.759,-118.474,60.833,-176.6541,-1.4916,0.0000
C01749=23.856,-115.434,60.496,-176.2287,-5.1072,0.0000
C01750=21.884,-111.053,59.862,-177.7620,-5.8906,0.0000
C01751=20.311,-106.271,58.595,-178.8138,-3.4384,0.0000
C01752=18.799,-102.037,56.970,179.4391,1.3661,0.0000
C01753=17.042,-98.929,55.416,172.9538,10.5519,0.0000
C01754=14.284,-97.259,54.299,147.2615,11.9753,0.0000
C01755=9.511,-97.093,53.857,141.2751,-1.2004,0.0000
C01756=4.729,-97.396,53.838,141.0478,-2.4582,0.0000
C01757=0.000,-97.513,53.851,141.0193,0.0002,0.0000
C01758=0.000,-97.513,53.851,141.0193,0.0002,0.0000
C01759=-4.728,-97.396,53.838,141.0478,2.4579,0.0000
C01760=-9.511,-97.093,53.857,141.2753,1.1983,0.0000
C01761=-14.284,-97.259,54.299,147.2610,-11.9745,0.0000
C01762=-17.042,-98.929,55.416,172.9538,-10.5519,0.0000
C01763=-18.799,-102.037,56.970,179.4391,-1.3661,0.0000
C01764=-20.311,-106.271,58.595,-178.8138,3.4384,0.0000
C01765=-21.884,-111.053,59.862,-177.7620,5.8906,0.0000
C01766=-23.856,-115.434,60.496,-176.2287,5.1072,0.0000
C01767=-27.759,-118.474,60.833,-176.6541,1.4916,0.0000
C01768=-33.133,-119.658,61.109,-177.9965,0.0483,0.0000
C01769=-39.003,-118.674,61.389,-179.8930,-0.0333,0.0000
C01770=-44.900,-116.647,61.575,-179.9867,-0.0050,0.0000
C01771=-50.733,-114.231,61.575,-179.9870,-0.0059,0.0000
C01772=-56.336,-111.494,61.389,-179.9008,-0.0521,0.0000
C01773=-61.183,-108.040,61.109,-178.6171,-1.4511,0.0000
C01774=-64.145,-103.402,60.833,-178.6866,-3.4195,0.0000
C01775=-64.755,-98.493,60.496,179.0498,-6.2664,0.0000
C01776=-63.051,-94.001,59.862,177.4051,-5.7440,0.0000
C01777=-60.783,-89.507,58.595,178.4051,-3.2696,0.0000
C01778=-58.858,-85.443,56.970,-179.4304,1.3626,0.0000
C01779=-57.903,-82.003,55.416,-177.4625,12.3592,0.0000
C01780=-58.672,-78.873,54.299,163.0569,31.1575,0.0000
C01781=-61.930,-75.380,53.857,149.8083,28.9069,0.0000
C01782=-65.526,-72.213,53.838,148.9527,28.4254,0.0000
C01783=-68.952,-68.952,53.851,150.2215,29.7787,0.0000
C01784=-72.213,-65.526,53.838,151.5744,31.0471,0.0000
C01785=-75.380,-61.930,53.857,151.0921,30.1904,0.0000
C01786=-78.873,-58.672,54.299,148.8426,16.9440,0.0000
C01787=-82.003,-57.903,55.416,167.6408,-2.5375,0.0000
C01788=-85.443,-58.858,56.970,178.6374,-0.5696,0.0000
C01789=-89.507,-60.783,58.595,-176.7304,1.5949,0.0000
C01790=-94.001,-63.051,59.862,-174.2560,2.5949,0.0000
C01791=-98.493,-64.755,60.496,-173.7336,0.9502,0.0000
C01792=-103.402,-64.145,60.833,-176.5805,-1.3134,0.0000
C01793=-108.040,-61.183,61.109,-178.5489,-1.3829,0.0000
C01794=-111.494,-56.336,61.389,-179.9479,-0.0992,0.0000
C01795=-114.231,-50.733,61.575,-179.9941,-0.0130,0.0000
C01796=-116.647,-44.900,61.575,-179.9950,-0.0133,0.0000
C01797=-118.674,-39.003,61.389,-179.9667,-0.1070,0.0000
C01798=-119.658,-33.133,61.109,179.9517,-2.0035,0.0000
C01799=-118.474,-27.759,60.833,178.5084,-3.3459,0.0000
C01800=-115.434,-23.856,60.496,174.8928,-3.7713,0.0000
C01801=-111.053,-21.884,59.862,174.1094,-2.2380,0.0000
C01802=-106.271,-20.311,58.595,176.5616,-1.1862,0.0000
C01803=-102.037,-18.799,56.970,-178.6339,0.5609,0.0000
C01804=-98.929,-17.042,55.416,-169.4481,7.0462,0.0000
C01805=-97.259,-14.284,54.299,-168.0247,32.7385,0.0000
C01806=-97.093,-9.511,53.857,178.7996,38.7249,0.0000
C01807=-97.396,-4.729,53.838,177.5418,38.9522,0.0000
C01808=-97.513,0.000,53.851,-179.9998,38.9807,0.0000
C01809=-97.396,4.728,53.838,-177.5421,38.9522,0.0000
C01810=-97.093,9.511,53.857,-178.8017,38.7247,0.0000
C01811=-97.259,14.284,54.299,168.0255,32.7390,0.0000
C01812=-98.929,17.042,55.416,169.4481,7.0462,0.0000
C01813=-102.037,18.799,56.970,178.6339,0.5609,0.0000
C01814=-106.271,20.311,58.595,-176.5616,-1.1862,0.0000
C01815=-111.053,21.884,59.862,-174.1094,-2.2380,0.0000
C01816=-115.434,23.856,60.496,-174.8928,-3.7713,0.0000
C01817=-118.474,27.759,60.833,-178.5084,-3.3459,0.0000
C01818=-119.658,33.133,61.109,-179.9517,-2.0035,0.0000
C01819=-118.674,39.003,61.389,179.9667,-0.1070,0.0000
C01820=-116.647,44.900,61.575,179.9950,-0.0133,0.0000
C01821=-114.231,50.733,61.575,179.9941,-0.0130,0.0000
C01822=-111.494,56.336,61.389,179.9479,-0.0992,0.0000
C01823=-108.040,61.183,61.109,178.5489,-1.3829,0.0000
C01824=-103.402,64.145,60.833,176.5805,-1.3134,0.0000
C01825=-98.493,64.755,60.496,173.7336,0.9502,0.0000
C01826=-94.001,63.051,59.862,174.2560,2.5949,0.0000
C01827=-89.507,60.783,58.595,176.7304,1.5949,0.0000
C01828=-85.443,58.858,56.970,-178.6374,-0.5696,0.0000
C01829=-82.003,57.903,55.416,-167.6408,-2.5375,0.0000
C01830=-78.873,58.672,54.299,-148.8425,16.9431,0.0000
C01831=-75.380,61.930,53.857,-151.0931,30.1917,0.0000
C01832=-72.213,65.526,53.838,-151.5746,31.0473,0.0000
C01833=-68.952,68.952,53.851,-150.2213,29.7785,0.0000
C01834=-65.526,72.213,53.838,-148.9529,28.4256,0.0000
C01835=-61.930,75.380,53.857,-149.8096,28.9079,0.0000
C01836=-58.672,78.873,54.299,-163.0560,31.1574,0.0000
C01837=-57.903,82.003,55.416,177.4625,12.3592,0.0000
C01838=-58.858,85.443,56.970,179.4304,1.3626,0.0000
C01839=-60.783,89.507,58.595,-178.4051,-3.2696,0.0000
C01840=-63.051,94.001,59.862,-177.4051,-5.7440,0.0000
C01841=-64.755,98.493,60.496,-179.0498,-6.2664,0.0000
C01842=-64.145,103.402,60.833,178.6866,-3.4195,0.0000
C01843=-61.183,108.040,61.109,178.6171,-1.4511,0.0000
C01844=-56.336,111.494,61.389,179.9008,-0.0521,0.0000
C01845=-50.733,114.231,61.575,179.9870,-0.0059,0.0000
C01846=-44.900,116.647,61.575,179.9867,-0.0050,0.0000
C01847=-39.003,118.674,61.389,179.8930,-0.0333,0.0000
C01848=-33.133,119.658,61.109,177.9965,0.0483,0.0000
C01849=-27.759,118.474,60.833,176.6541,1.4916,0.0000
C01850=-23.856,115.434,60.496,176.2287,5.1072,0.0000
